LIN {X 0,Y 223.489,Z 613.022,A -85,B 0,C 180,E1 -23403.605,E2 -23403.605} C_VEL
LIN {X 0,Y 223.354,Z 613.371,A -85,B 0,C 180,E1 -23409.051,E2 -23409.051} C_VEL
LIN {X 0,Y 224.233,Z 615.221,A -85,B 0,C 180,E1 -23413.695,E2 -23413.695} C_VEL
LIN {X 0,Y 226.542,Z 620.688,A -85,B 0,C 180,E1 -23419.952,E2 -23419.952} C_VEL
LIN {X 0,Y 227.439,Z 623.666,A -85,B 0,C 180,E1 -23422.032,E2 -23422.032} C_VEL
LIN {X 0,Y 228.456,Z 630.685,A -85,B 0,C 180,E1 -23425.51,E2 -23425.51} C_VEL
LIN {X 0,Y 229.459,Z 640.943,A -85,B 0,C 180,E1 -23429.676,E2 -23429.676} C_VEL
LIN {X 0,Y 229.456,Z 644.838,A -85,B 0,C 180,E1 -23430.955,E2 -23430.955} C_VEL
LIN {X 0,Y 226.429,Z 656.895,A -85,B 0,C 180,E1 -23433.683,E2 -23433.683} C_VEL
LIN {X 0,Y 221.885,Z 669.855,A -85,B 0,C 180,E1 -23436.516,E2 -23436.516} C_VEL
LIN {X 0,Y 214.485,Z 681.955,A -85,B 0,C 180,E1 -23438.563,E2 -23438.563} C_VEL
LIN {X 0,Y 205.907,Z 694.618,A -85,B 0,C 180,E1 -23441.336,E2 -23441.336} C_VEL
LIN {X 0,Y 198.409,Z 704.732,A -85,B 0,C 180,E1 -23444.173,E2 -23444.173} C_VEL
LIN {X 0,Y 190.475,Z 714.65,A -85,B 0,C 180,E1 -23447.682,E2 -23447.682} C_VEL
LIN {X 0,Y 184.311,Z 722.053,A -85,B 0,C 180,E1 -23451.015,E2 -23451.015} C_VEL
LIN {X 0,Y 178.043,Z 729.213,A -85,B 0,C 180,E1 -23455.088,E2 -23455.088} C_VEL
LIN {X 0,Y 172.781,Z 735.226,A -85,B 0,C 180,E1 -23459.443,E2 -23459.443} C_VEL
LIN {X 0,Y 167.694,Z 741.138,A -85,B 0,C 180,E1 -23465.226,E2 -23465.226} C_VEL
LIN {X 0,Y 164.518,Z 745.056,A -85,B 0,C 180,E1 -23470.746,E2 -23470.746} C_VEL
LIN {X 0,Y 163.031,Z 746.186,A -85,B 0,C 180,E1 -23472.711,E2 -23472.711} C_VEL
LIN {X 0,Y 159.183,Z 747.539,A -85,B 0,C 180,E1 -23475.926,E2 -23475.926} C_VEL
LIN {X 0,Y 156.295,Z 748.29,A -85,B 0,C 180,E1 -23478.609,E2 -23478.609} C_VEL
LIN {X 0,Y 155.1,Z 748.716,A -85,B 0,C 180,E1 -23480.741,E2 -23480.741} C_VEL
LIN {X 0,Y 155.005,Z 748.773,A -85,B 0,C 180,E1 -23481.468,E2 -23481.468} C_VEL
LIN {X 0,Y 155.163,Z 749.11,A -85,B 0,C 180,E1 -23485.174,E2 -23485.174} C_VEL
LIN {X 0,Y 155.407,Z 748.7,A -85,B 0,C 180,E1 -23490.003,E2 -23490.003} C_VEL
LIN {X 0,Y 155.267,Z 747.247,A -85,B 0,C 180,E1 -23495.262,E2 -23495.262} C_VEL
LIN {X 0,Y 155.222,Z 744.685,A -85,B 0,C 180,E1 -23500.437,E2 -23500.437} C_VEL
LIN {X 0,Y 156.163,Z 741.06,A -85,B 0,C 180,E1 -23505.668,E2 -23505.668} C_VEL
LIN {X 0,Y 158.061,Z 736.145,A -85,B 0,C 180,E1 -23510.977,E2 -23510.977} C_VEL
LIN {X 0,Y 160.289,Z 731.655,A -85,B 0,C 180,E1 -23514.965,E2 -23514.965} C_VEL
LIN {X 0,Y 165.09,Z 728.65,A -85,B 0,C 180,E1 -23520.723,E2 -23520.723} C_VEL
LIN {X 0,Y 173.61,Z 723.828,A -85,B 0,C 180,E1 -23527.392,E2 -23527.392} C_VEL
LIN {X 0,Y 186.812,Z 716.879,A -85,B 0,C 180,E1 -23534.108,E2 -23534.108} C_VEL
LIN {X 0,Y 199.391,Z 710.477,A -85,B 0,C 180,E1 -23538.657,E2 -23538.657} C_VEL
LIN {X 0,Y 200.155,Z 709.902,A -85,B 0,C 180,E1 -23539.319,E2 -23539.319} C_VEL
LIN {X 0,Y 189.134,Z 711.932,A -85,B 0,C 180,E1 -23543.521,E2 -23543.521} C_VEL
LIN {X 0,Y 178.051,Z 713.204,A -85,B 0,C 180,E1 -23549.128,E2 -23549.128} C_VEL
LIN {X 0,Y 169.257,Z 713.167,A -85,B 0,C 180,E1 -23555.468,E2 -23555.468} C_VEL
LIN {X 0,Y 162.754,Z 711.681,A -85,B 0,C 180,E1 -23562.407,E2 -23562.407} C_VEL
LIN {X 0,Y 159.866,Z 709.778,A -85,B 0,C 180,E1 -23567.303,E2 -23567.303} C_VEL
LIN {X 0,Y 157.754,Z 707.203,A -85,B 0,C 180,E1 -23572.321,E2 -23572.321} C_VEL
LIN {X 0,Y 156.22,Z 701.701,A -85,B 0,C 180,E1 -23580.001,E2 -23580.001} C_VEL
LIN {X 0,Y 156.351,Z 696.898,A -85,B 0,C 180,E1 -23585.159,E2 -23585.159} C_VEL
LIN {X 0,Y 156.849,Z 691.072,A -85,B 0,C 180,E1 -23590.326,E2 -23590.326} C_VEL
LIN {X 0,Y 158.04,Z 684.129,A -85,B 0,C 180,E1 -23595.476,E2 -23595.476} C_VEL
LIN {X 0,Y 160.485,Z 674.694,A -85,B 0,C 180,E1 -23601.18,E2 -23601.18} C_VEL
LIN {X 0,Y 164.064,Z 663.436,A -85,B 0,C 180,E1 -23606.731,E2 -23606.731} C_VEL
LIN {X 0,Y 168.255,Z 651.541,A -85,B 0,C 180,E1 -23611.476,E2 -23611.476} C_VEL
LIN {X 0,Y 173.138,Z 637.728,A -85,B 0,C 180,E1 -23615.982,E2 -23615.982} C_VEL
LIN {X 0,Y 178.436,Z 623.245,A -85,B 0,C 180,E1 -23619.796,E2 -23619.796} C_VEL
LIN {X 0,Y 180.247,Z 618.116,A -85,B 0,C 180,E1 -23620.962,E2 -23620.962} C_VEL
LIN {X 0,Y 180.924,Z 618.131,A -85,B 0,C 180,E1 -23621.329,E2 -23621.329} C_VEL
LIN {X 0,Y 183.088,Z 617.315,A -85,B 0,C 180,E1 -23622.204,E2 -23622.204} C_VEL
LIN {X 0,Y 185.677,Z 615.473,A -85,B 0,C 180,E1 -23622.948,E2 -23622.948} C_VEL
LIN {X 0,Y 189.612,Z 611.812,A -85,B 0,C 180,E1 -23623.859,E2 -23623.859} C_VEL
LIN {X 0,Y 191.1,Z 610.979,A -85,B 0,C 180,E1 -23624.328,E2 -23624.328} C_VEL
LIN {X 0,Y 200.001,Z 609.038,A -85,B 0,C 180,E1 -23627.557,E2 -23627.557} C_VEL
LIN {X 0,Y 202.173,Z 618.005,A -85,B 0,C 180,E1 -23630.328,E2 -23630.328} C_VEL
LIN {X 0,Y 203.073,Z 626.979,A -85,B 0,C 180,E1 -23632.75,E2 -23632.75} C_VEL
LIN {X 0,Y 203.116,Z 633.014,A -85,B 0,C 180,E1 -23634.296,E2 -23634.296} C_VEL
LIN {X 0,Y 197.422,Z 646.866,A -85,B 0,C 180,E1 -23636.508,E2 -23636.508} C_VEL
LIN {X 0,Y 191.451,Z 659.757,A -85,B 0,C 180,E1 -23639.072,E2 -23639.072} C_VEL
LIN {X 0,Y 185.064,Z 672.439,A -85,B 0,C 180,E1 -23642.274,E2 -23642.274} C_VEL
LIN {X 0,Y 179.25,Z 683.136,A -85,B 0,C 180,E1 -23645.687,E2 -23645.687} C_VEL
LIN {X 0,Y 173.819,Z 692.349,A -85,B 0,C 180,E1 -23649.278,E2 -23649.278} C_VEL
LIN {X 0,Y 169.275,Z 700.275,A -85,B 0,C 180,E1 -23653.102,E2 -23653.102} C_VEL
LIN {X 0,Y 164.71,Z 707.873,A -85,B 0,C 180,E1 -23657.679,E2 -23657.679} C_VEL
LIN {X 0,Y 161.077,Z 714.188,A -85,B 0,C 180,E1 -23662.476,E2 -23662.476} C_VEL
LIN {X 0,Y 158.265,Z 719.384,A -85,B 0,C 180,E1 -23667.452,E2 -23667.452} C_VEL
LIN {X 0,Y 156.429,Z 723.388,A -85,B 0,C 180,E1 -23672.572,E2 -23672.572} C_VEL
LIN {X 0,Y 155.289,Z 726.446,A -85,B 0,C 180,E1 -23677.8,E2 -23677.8} C_VEL
LIN {X 0,Y 154.783,Z 728.481,A -85,B 0,C 180,E1 -23683.119,E2 -23683.119} C_VEL
LIN {X 0,Y 154.975,Z 729.558,A -85,B 0,C 180,E1 -23688.505,E2 -23688.505} C_VEL
LIN {X 0,Y 155.836,Z 729.668,A -85,B 0,C 180,E1 -23693.943,E2 -23693.943} C_VEL
LIN {X 0,Y 157.571,Z 728.723,A -85,B 0,C 180,E1 -23699.378,E2 -23699.378} C_VEL
LIN {X 0,Y 160.35,Z 726.79,A -85,B 0,C 180,E1 -23704.731,E2 -23704.731} C_VEL
LIN {X 0,Y 164.191,Z 723.669,A -85,B 0,C 180,E1 -23709.941,E2 -23709.941} C_VEL
LIN {X 0,Y 169.393,Z 719.182,A -85,B 0,C 180,E1 -23715.143,E2 -23715.143} C_VEL
LIN {X 0,Y 175.246,Z 713.903,A -85,B 0,C 180,E1 -23719.633,E2 -23719.633} C_VEL
LIN {X 0,Y 182.399,Z 706.964,A -85,B 0,C 180,E1 -23724.008,E2 -23724.008} C_VEL
LIN {X 0,Y 189.42,Z 699.593,A -85,B 0,C 180,E1 -23727.569,E2 -23727.569} C_VEL
LIN {X 0,Y 197.066,Z 690.909,A -85,B 0,C 180,E1 -23730.892,E2 -23730.892} C_VEL
LIN {X 0,Y 205.336,Z 680.628,A -85,B 0,C 180,E1 -23733.949,E2 -23733.949} C_VEL
LIN {X 0,Y 214.102,Z 668.356,A -85,B 0,C 180,E1 -23736.79,E2 -23736.79} C_VEL
LIN {X 0,Y 221.298,Z 656.932,A -85,B 0,C 180,E1 -23738.883,E2 -23738.883} C_VEL
LIN {X 0,Y 225.042,Z 650.417,A -85,B 0,C 180,E1 -23739.907,E2 -23739.907} C_VEL
LIN {X 0,Y 225.084,Z 646.05,A -85,B 0,C 180,E1 -23741.805,E2 -23741.805} C_VEL
LIN {X 0,Y 224.673,Z 640.373,A -85,B 0,C 180,E1 -23744.579,E2 -23744.579} C_VEL
LIN {X 0,Y 223.711,Z 634.018,A -85,B 0,C 180,E1 -23748.216,E2 -23748.216} C_VEL
LIN {X 0,Y 222.644,Z 628.828,A -85,B 0,C 180,E1 -23751.833,E2 -23751.833} C_VEL
LIN {X 0,Y 221.481,Z 623.917,A -85,B 0,C 180,E1 -23756.361,E2 -23756.361} C_VEL
LIN {X 0,Y 220.778,Z 621.33,A -85,B 0,C 180,E1 -23759.999,E2 -23759.999} C_VEL
LIN {X 0,Y 220.569,Z 619.485,A -85,B 0,C 180,E1 -23763.653,E2 -23763.653} C_VEL
LIN {X 0,Y 220.459,Z 619.877,A -85,B 0,C 180,E1 -23769.171,E2 -23769.171} C_VEL
LIN {X 0,Y 221.087,Z 621.231,A -85,B 0,C 180,E1 -23772.856,E2 -23772.856} C_VEL
LIN {X 0,Y 222.002,Z 624.081,A -85,B 0,C 180,E1 -23776.553,E2 -23776.553} C_VEL
LIN {X 0,Y 223.485,Z 627.57,A -85,B 0,C 180,E1 -23780.237,E2 -23780.237} C_VEL
LIN {X 0,Y 223.819,Z 628.846,A -85,B 0,C 180,E1 -23781.167,E2 -23781.167} C_VEL
LIN {X 0,Y 224.544,Z 635.94,A -85,B 0,C 180,E1 -23784.821,E2 -23784.821} C_VEL
LIN {X 0,Y 225.046,Z 644.518,A -85,B 0,C 180,E1 -23788.484,E2 -23788.484} C_VEL
LIN {X 0,Y 225.04,Z 647.083,A -85,B 0,C 180,E1 -23789.463,E2 -23789.463} C_VEL
LIN {X 0,Y 224.83,Z 648.862,A -85,B 0,C 180,E1 -23790.009,E2 -23790.009} C_VEL
LIN {X 0,Y 221.559,Z 660.162,A -85,B 0,C 180,E1 -23792.632,E2 -23792.632} C_VEL
LIN {X 0,Y 217.114,Z 671.412,A -85,B 0,C 180,E1 -23795.185,E2 -23795.185} C_VEL
LIN {X 0,Y 209.21,Z 683.673,A -85,B 0,C 180,E1 -23797.321,E2 -23797.321} C_VEL
LIN {X 0,Y 201.277,Z 694.886,A -85,B 0,C 180,E1 -23799.814,E2 -23799.814} C_VEL
LIN {X 0,Y 193.488,Z 704.878,A -85,B 0,C 180,E1 -23802.652,E2 -23802.652} C_VEL
LIN {X 0,Y 185.57,Z 714.288,A -85,B 0,C 180,E1 -23806.018,E2 -23806.018} C_VEL
LIN {X 0,Y 178.802,Z 722.034,A -85,B 0,C 180,E1 -23809.572,E2 -23809.572} C_VEL
LIN {X 0,Y 170.689,Z 730.731,A -85,B 0,C 180,E1 -23814.803,E2 -23814.803} C_VEL
LIN {X 0,Y 164.249,Z 737.577,A -85,B 0,C 180,E1 -23820.527,E2 -23820.527} C_VEL
LIN {X 0,Y 159.501,Z 742.743,A -85,B 0,C 180,E1 -23826.64,E2 -23826.64} C_VEL
LIN {X 0,Y 156.926,Z 745.738,A -85,B 0,C 180,E1 -23831.733,E2 -23831.733} C_VEL
LIN {X 0,Y 155.418,Z 747.806,A -85,B 0,C 180,E1 -23836.935,E2 -23836.935} C_VEL
LIN {X 0,Y 155.005,Z 748.773,A -85,B 0,C 180,E1 -23841.468,E2 -23841.468} C_VEL
LIN {X 0,Y 154.379,Z 749.017,A -85,B 0,C 180,E1 -23843.64,E2 -23843.64} C_VEL
LIN {X 0,Y 152.898,Z 748.974,A -85,B 0,C 180,E1 -23845.787,E2 -23845.787} C_VEL
LIN {X 0,Y 148.562,Z 747.904,A -85,B 0,C 180,E1 -23851.659,E2 -23851.659} C_VEL
LIN {X 0,Y 148.205,Z 747.43,A -85,B 0,C 180,E1 -23853.196,E2 -23853.196} C_VEL
LIN {X 0,Y 148.17,Z 746.707,A -85,B 0,C 180,E1 -23855.446,E2 -23855.446} C_VEL
LIN {X 0,Y 148.186,Z 744.082,A -85,B 0,C 180,E1 -23860.938,E2 -23860.938} C_VEL
LIN {X 0,Y 149.659,Z 739.281,A -85,B 0,C 180,E1 -23867.775,E2 -23867.775} C_VEL
LIN {X 0,Y 151.942,Z 734.123,A -85,B 0,C 180,E1 -23873.154,E2 -23873.154} C_VEL
LIN {X 0,Y 153.762,Z 730.941,A -85,B 0,C 180,E1 -23876.102,E2 -23876.102} C_VEL
LIN {X 0,Y 161.607,Z 726.826,A -85,B 0,C 180,E1 -23884.429,E2 -23884.429} C_VEL
LIN {X 0,Y 171.546,Z 722.041,A -85,B 0,C 180,E1 -23890.96,E2 -23890.96} C_VEL
LIN {X 0,Y 184.2,Z 716.172,A -85,B 0,C 180,E1 -23896.626,E2 -23896.626} C_VEL
LIN {X 0,Y 190.089,Z 713.503,A -85,B 0,C 180,E1 -23898.714,E2 -23898.714} C_VEL
LIN {X 0,Y 190.869,Z 712.92,A -85,B 0,C 180,E1 -23899.48,E2 -23899.48} C_VEL
LIN {X 0,Y 179.634,Z 714.285,A -85,B 0,C 180,E1 -23904.067,E2 -23904.067} C_VEL
LIN {X 0,Y 168.819,Z 714.719,A -85,B 0,C 180,E1 -23910.03,E2 -23910.03} C_VEL
LIN {X 0,Y 160.341,Z 713.845,A -85,B 0,C 180,E1 -23916.767,E2 -23916.767} C_VEL
LIN {X 0,Y 154.361,Z 711.482,A -85,B 0,C 180,E1 -23924.148,E2 -23924.148} C_VEL
LIN {X 0,Y 151.752,Z 709.006,A -85,B 0,C 180,E1 -23929.326,E2 -23929.326} C_VEL
LIN {X 0,Y 149.904,Z 705.812,A -85,B 0,C 180,E1 -23934.621,E2 -23934.621} C_VEL
LIN {X 0,Y 149.08,Z 700.566,A -85,B 0,C 180,E1 -23941.352,E2 -23941.352} C_VEL
LIN {X 0,Y 149.332,Z 695.303,A -85,B 0,C 180,E1 -23946.758,E2 -23946.758} C_VEL
LIN {X 0,Y 150.076,Z 689,A -85,B 0,C 180,E1 -23952.167,E2 -23952.167} C_VEL
LIN {X 0,Y 151.833,Z 680.442,A -85,B 0,C 180,E1 -23958.208,E2 -23958.208} C_VEL
LIN {X 0,Y 154.571,Z 671.347,A -85,B 0,C 180,E1 -23963.445,E2 -23963.445} C_VEL
LIN {X 0,Y 158.134,Z 660.693,A -85,B 0,C 180,E1 -23968.541,E2 -23968.541} C_VEL
LIN {X 0,Y 162.689,Z 648.26,A -85,B 0,C 180,E1 -23973.422,E2 -23973.422} C_VEL
LIN {X 0,Y 167.242,Z 635.959,A -85,B 0,C 180,E1 -23977.391,E2 -23977.391} C_VEL
LIN {X 0,Y 169.446,Z 630.318,A -85,B 0,C 180,E1 -23979.046,E2 -23979.046} C_VEL
LIN {X 0,Y 170.577,Z 630.187,A -85,B 0,C 180,E1 -23979.69,E2 -23979.69} C_VEL
LIN {X 0,Y 172.808,Z 629.111,A -85,B 0,C 180,E1 -23980.597,E2 -23980.597} C_VEL
LIN {X 0,Y 176.713,Z 626.375,A -85,B 0,C 180,E1 -23981.773,E2 -23981.773} C_VEL
LIN {X 0,Y 178.152,Z 625.177,A -85,B 0,C 180,E1 -23982.118,E2 -23982.118} C_VEL
LIN {X 0,Y 183.046,Z 622.498,A -85,B 0,C 180,E1 -23983.719,E2 -23983.719} C_VEL
LIN {X 0,Y 187.136,Z 619.45,A -85,B 0,C 180,E1 -23984.764,E2 -23984.764} C_VEL
LIN {X 0,Y 188.591,Z 618.221,A -85,B 0,C 180,E1 -23985.078,E2 -23985.078} C_VEL
LIN {X 0,Y 193.37,Z 616.385,A -85,B 0,C 180,E1 -23986.628,E2 -23986.628} C_VEL
LIN {X 0,Y 195.642,Z 615.928,A -85,B 0,C 180,E1 -23987.428,E2 -23987.428} C_VEL
LIN {X 0,Y 196.622,Z 619.354,A -85,B 0,C 180,E1 -23988.645,E2 -23988.645} C_VEL
LIN {X 0,Y 197.469,Z 625.794,A -85,B 0,C 180,E1 -23990.579,E2 -23990.579} C_VEL
LIN {X 0,Y 197.745,Z 633.888,A -85,B 0,C 180,E1 -23992.827,E2 -23992.827} C_VEL
LIN {X 0,Y 196.896,Z 636.565,A -85,B 0,C 180,E1 -23993.28,E2 -23993.28} C_VEL
LIN {X 0,Y 190.573,Z 651.082,A -85,B 0,C 180,E1 -23995.776,E2 -23995.776} C_VEL
LIN {X 0,Y 184.485,Z 663.343,A -85,B 0,C 180,E1 -23998.41,E2 -23998.41} C_VEL
LIN {X 0,Y 177.966,Z 675.514,A -85,B 0,C 180,E1 -24001.711,E2 -24001.711} C_VEL
LIN {X 0,Y 172.001,Z 685.898,A -85,B 0,C 180,E1 -24005.238,E2 -24005.238} C_VEL
LIN {X 0,Y 165.764,Z 695.986,A -85,B 0,C 180,E1 -24009.524,E2 -24009.524} C_VEL
LIN {X 0,Y 161.111,Z 703.593,A -85,B 0,C 180,E1 -24013.68,E2 -24013.68} C_VEL
LIN {X 0,Y 156.765,Z 710.557,A -85,B 0,C 180,E1 -24018.359,E2 -24018.359} C_VEL
LIN {X 0,Y 153.221,Z 716.506,A -85,B 0,C 180,E1 -24023.413,E2 -24023.413} C_VEL
LIN {X 0,Y 150.114,Z 722.307,A -85,B 0,C 180,E1 -24029.997,E2 -24029.997} C_VEL
LIN {X 0,Y 148.488,Z 726.191,A -85,B 0,C 180,E1 -24036.3,E2 -24036.3} C_VEL
LIN {X 0,Y 147.829,Z 728.225,A -85,B 0,C 180,E1 -24040.959,E2 -24040.959} C_VEL
LIN {X 0,Y 147.753,Z 729.674,A -85,B 0,C 180,E1 -24046.579,E2 -24046.579} C_VEL
LIN {X 0,Y 148.348,Z 730.206,A -85,B 0,C 180,E1 -24052.268,E2 -24052.268} C_VEL
LIN {X 0,Y 149.877,Z 729.71,A -85,B 0,C 180,E1 -24057.961,E2 -24057.961} C_VEL
LIN {X 0,Y 152.731,Z 727.977,A -85,B 0,C 180,E1 -24064.076,E2 -24064.076} C_VEL
LIN {X 0,Y 156.109,Z 725.6,A -85,B 0,C 180,E1 -24069.066,E2 -24069.066} C_VEL
LIN {X 0,Y 162.176,Z 720.844,A -85,B 0,C 180,E1 -24075.44,E2 -24075.44} C_VEL
LIN {X 0,Y 168.647,Z 715.369,A -85,B 0,C 180,E1 -24080.434,E2 -24080.434} C_VEL
LIN {X 0,Y 176.015,Z 708.671,A -85,B 0,C 180,E1 -24084.933,E2 -24084.933} C_VEL
LIN {X 0,Y 184.328,Z 700.456,A -85,B 0,C 180,E1 -24089.073,E2 -24089.073} C_VEL
LIN {X 0,Y 192.282,Z 691.867,A -85,B 0,C 180,E1 -24092.412,E2 -24092.412} C_VEL
LIN {X 0,Y 200.84,Z 681.65,A -85,B 0,C 180,E1 -24095.474,E2 -24095.474} C_VEL
LIN {X 0,Y 208.184,Z 671.874,A -85,B 0,C 180,E1 -24097.794,E2 -24097.794} C_VEL
LIN {X 0,Y 215.952,Z 660.423,A -85,B 0,C 180,E1 -24099.996,E2 -24099.996} C_VEL
LIN {X 0,Y 219.532,Z 654.659,A -85,B 0,C 180,E1 -24100.938,E2 -24100.938} C_VEL
LIN {X 0,Y 220.2,Z 652.915,A -85,B 0,C 180,E1 -24101.387,E2 -24101.387} C_VEL
LIN {X 0,Y 220.25,Z 647.016,A -85,B 0,C 180,E1 -24104.262,E2 -24104.262} C_VEL
LIN {X 0,Y 219.848,Z 642.047,A -85,B 0,C 180,E1 -24107.068,E2 -24107.068} C_VEL
LIN {X 0,Y 219.123,Z 636.488,A -85,B 0,C 180,E1 -24110.771,E2 -24110.771} C_VEL
LIN {X 0,Y 218.552,Z 633.135,A -85,B 0,C 180,E1 -24113.537,E2 -24113.537} C_VEL
LIN {X 0,Y 218.036,Z 630.331,A -85,B 0,C 180,E1 -24116.303,E2 -24116.303} C_VEL
LIN {X 0,Y 217.543,Z 627.695,A -85,B 0,C 180,E1 -24119.999,E2 -24119.999} C_VEL
LIN {X 0,Y 217.4,Z 625.859,A -85,B 0,C 180,E1 -24123.706,E2 -24123.706} C_VEL
LIN {X 0,Y 217.358,Z 626.302,A -85,B 0,C 180,E1 -24129.303,E2 -24129.303} C_VEL
LIN {X 0,Y 217.941,Z 627.789,A -85,B 0,C 180,E1 -24133.045,E2 -24133.045} C_VEL
LIN {X 0,Y 218.808,Z 630.672,A -85,B 0,C 180,E1 -24136.802,E2 -24136.802} C_VEL
LIN {X 0,Y 219.727,Z 632.927,A -85,B 0,C 180,E1 -24139.256,E2 -24139.256} C_VEL
LIN {X 0,Y 220.142,Z 634.473,A -85,B 0,C 180,E1 -24140.558,E2 -24140.558} C_VEL
LIN {X 0,Y 220.49,Z 640.824,A -85,B 0,C 180,E1 -24143.978,E2 -24143.978} C_VEL
LIN {X 0,Y 220.592,Z 649.938,A -85,B 0,C 180,E1 -24148.028,E2 -24148.028} C_VEL
LIN {X 0,Y 220.209,Z 652.857,A -85,B 0,C 180,E1 -24149.028,E2 -24149.028} C_VEL
LIN {X 0,Y 216.478,Z 663.697,A -85,B 0,C 180,E1 -24151.632,E2 -24151.632} C_VEL
LIN {X 0,Y 212.462,Z 672.993,A -85,B 0,C 180,E1 -24153.792,E2 -24153.792} C_VEL
LIN {X 0,Y 204.686,Z 684.456,A -85,B 0,C 180,E1 -24155.827,E2 -24155.827} C_VEL
LIN {X 0,Y 196.796,Z 695.125,A -85,B 0,C 180,E1 -24158.222,E2 -24158.222} C_VEL
LIN {X 0,Y 187.623,Z 706.369,A -85,B 0,C 180,E1 -24161.486,E2 -24161.486} C_VEL
LIN {X 0,Y 179.119,Z 715.833,A -85,B 0,C 180,E1 -24165.073,E2 -24165.073} C_VEL
LIN {X 0,Y 171.525,Z 723.841,A -85,B 0,C 180,E1 -24169.04,E2 -24169.04} C_VEL
LIN {X 0,Y 164.864,Z 730.604,A -85,B 0,C 180,E1 -24173.362,E2 -24173.362} C_VEL
LIN {X 0,Y 157.986,Z 737.372,A -85,B 0,C 180,E1 -24179.235,E2 -24179.235} C_VEL
LIN {X 0,Y 152.895,Z 742.475,A -85,B 0,C 180,E1 -24185.566,E2 -24185.566} C_VEL
LIN {X 0,Y 150.109,Z 745.398,A -85,B 0,C 180,E1 -24190.872,E2 -24190.872} C_VEL
LIN {X 0,Y 148.425,Z 747.432,A -85,B 0,C 180,E1 -24196.308,E2 -24196.308} C_VEL
LIN {X 0,Y 147.935,Z 748.453,A -85,B 0,C 180,E1 -24201.809,E2 -24201.809} C_VEL
LIN {X 0,Y 148.08,Z 748.629,A -85,B 0,C 180,E1 -24205.315,E2 -24205.315} C_VEL
LIN {X 0,Y 148.34,Z 748.202,A -85,B 0,C 180,E1 -24210.003,E2 -24210.003} C_VEL
LIN {X 0,Y 148.205,Z 747.43,A -85,B 0,C 180,E1 -24213.196,E2 -24213.196} C_VEL
LIN {X 0,Y 147.436,Z 746.663,A -85,B 0,C 180,E1 -24215.438,E2 -24215.438} C_VEL
LIN {X 0,Y 144.551,Z 744.902,A -85,B 0,C 180,E1 -24219.095,E2 -24219.095} C_VEL
LIN {X 0,Y 142.342,Z 743.201,A -85,B 0,C 180,E1 -24222.094,E2 -24222.094} C_VEL
LIN {X 0,Y 141.682,Z 741.692,A -85,B 0,C 180,E1 -24224.414,E2 -24224.414} C_VEL
LIN {X 0,Y 141.778,Z 741.182,A -85,B 0,C 180,E1 -24225.192,E2 -24225.192} C_VEL
LIN {X 0,Y 143.322,Z 737.404,A -85,B 0,C 180,E1 -24230.078,E2 -24230.078} C_VEL
LIN {X 0,Y 146.163,Z 731.888,A -85,B 0,C 180,E1 -24235.645,E2 -24235.645} C_VEL
LIN {X 0,Y 147.333,Z 730.153,A -85,B 0,C 180,E1 -24237.334,E2 -24237.334} C_VEL
LIN {X 0,Y 154.789,Z 726.854,A -85,B 0,C 180,E1 -24245.19,E2 -24245.19} C_VEL
LIN {X 0,Y 166.205,Z 721.991,A -85,B 0,C 180,E1 -24252.578,E2 -24252.578} C_VEL
LIN {X 0,Y 180.789,Z 716.05,A -85,B 0,C 180,E1 -24258.769,E2 -24258.769} C_VEL
LIN {X 0,Y 181.54,Z 715.474,A -85,B 0,C 180,E1 -24259.647,E2 -24259.647} C_VEL
LIN {X 0,Y 170.099,Z 716.149,A -85,B 0,C 180,E1 -24264.66,E2 -24264.66} C_VEL
LIN {X 0,Y 162.82,Z 716.042,A -85,B 0,C 180,E1 -24268.805,E2 -24268.805} C_VEL
LIN {X 0,Y 153.899,Z 714.772,A -85,B 0,C 180,E1 -24275.734,E2 -24275.734} C_VEL
LIN {X 0,Y 149.359,Z 713.166,A -85,B 0,C 180,E1 -24280.77,E2 -24280.77} C_VEL
LIN {X 0,Y 144.787,Z 709.4,A -85,B 0,C 180,E1 -24288.806,E2 -24288.806} C_VEL
LIN {X 0,Y 142.299,Z 703.903,A -85,B 0,C 180,E1 -24297.17,E2 -24297.17} C_VEL
LIN {X 0,Y 142.115,Z 697.855,A -85,B 0,C 180,E1 -24304.255,E2 -24304.255} C_VEL
LIN {X 0,Y 142.819,Z 690.204,A -85,B 0,C 180,E1 -24311.353,E2 -24311.353} C_VEL
LIN {X 0,Y 144.486,Z 681.679,A -85,B 0,C 180,E1 -24317.7,E2 -24317.7} C_VEL
LIN {X 0,Y 147.108,Z 672.694,A -85,B 0,C 180,E1 -24323.214,E2 -24323.214} C_VEL
LIN {X 0,Y 150.757,Z 662.199,A -85,B 0,C 180,E1 -24328.546,E2 -24328.546} C_VEL
LIN {X 0,Y 155.392,Z 649.876,A -85,B 0,C 180,E1 -24333.646,E2 -24333.646} C_VEL
LIN {X 0,Y 158.706,Z 641.127,A -85,B 0,C 180,E1 -24336.789,E2 -24336.789} C_VEL
LIN {X 0,Y 160.394,Z 640.817,A -85,B 0,C 180,E1 -24337.84,E2 -24337.84} C_VEL
LIN {X 0,Y 162.587,Z 639.739,A -85,B 0,C 180,E1 -24338.814,E2 -24338.814} C_VEL
LIN {X 0,Y 167.748,Z 636.226,A -85,B 0,C 180,E1 -24340.497,E2 -24340.497} C_VEL
LIN {X 0,Y 169.961,Z 635.352,A -85,B 0,C 180,E1 -24341.424,E2 -24341.424} C_VEL
LIN {X 0,Y 172.386,Z 634.118,A -85,B 0,C 180,E1 -24342.276,E2 -24342.276} C_VEL
LIN {X 0,Y 176.477,Z 631.399,A -85,B 0,C 180,E1 -24343.392,E2 -24343.392} C_VEL
LIN {X 0,Y 177.913,Z 630.272,A -85,B 0,C 180,E1 -24343.734,E2 -24343.734} C_VEL
LIN {X 0,Y 182.982,Z 627.571,A -85,B 0,C 180,E1 -24345.281,E2 -24345.281} C_VEL
LIN {X 0,Y 188.642,Z 623.693,A -85,B 0,C 180,E1 -24346.594,E2 -24346.594} C_VEL
LIN {X 0,Y 191.092,Z 622.815,A -85,B 0,C 180,E1 -24347.356,E2 -24347.356} C_VEL
LIN {X 0,Y 191.778,Z 624.167,A -85,B 0,C 180,E1 -24348.016,E2 -24348.016} C_VEL
LIN {X 0,Y 192.285,Z 631.101,A -85,B 0,C 180,E1 -24350.136,E2 -24350.136} C_VEL
LIN {X 0,Y 192.307,Z 636.049,A -85,B 0,C 180,E1 -24351.588,E2 -24351.588} C_VEL
LIN {X 0,Y 186.942,Z 648.413,A -85,B 0,C 180,E1 -24353.691,E2 -24353.691} C_VEL
LIN {X 0,Y 180.544,Z 661.203,A -85,B 0,C 180,E1 -24356.307,E2 -24356.307} C_VEL
LIN {X 0,Y 174.638,Z 672.113,A -85,B 0,C 180,E1 -24359.127,E2 -24359.127} C_VEL
LIN {X 0,Y 168.256,Z 683.004,A -85,B 0,C 180,E1 -24362.645,E2 -24362.645} C_VEL
LIN {X 0,Y 162.281,Z 692.393,A -85,B 0,C 180,E1 -24366.382,E2 -24366.382} C_VEL
LIN {X 0,Y 157.102,Z 700.423,A -85,B 0,C 180,E1 -24370.394,E2 -24370.394} C_VEL
LIN {X 0,Y 152.019,Z 708.15,A -85,B 0,C 180,E1 -24375.267,E2 -24375.267} C_VEL
LIN {X 0,Y 147.88,Z 714.597,A -85,B 0,C 180,E1 -24380.422,E2 -24380.422} C_VEL
LIN {X 0,Y 144.692,Z 719.857,A -85,B 0,C 180,E1 -24385.819,E2 -24385.819} C_VEL
LIN {X 0,Y 142.987,Z 723.08,A -85,B 0,C 180,E1 -24389.997,E2 -24389.997} C_VEL
LIN {X 0,Y 141.399,Z 726.686,A -85,B 0,C 180,E1 -24396.233,E2 -24396.233} C_VEL
LIN {X 0,Y 140.676,Z 728.817,A -85,B 0,C 180,E1 -24401.524,E2 -24401.524} C_VEL
LIN {X 0,Y 140.729,Z 730.218,A -85,B 0,C 180,E1 -24407.432,E2 -24407.432} C_VEL
LIN {X 0,Y 141.465,Z 730.65,A -85,B 0,C 180,E1 -24413.415,E2 -24413.415} C_VEL
LIN {X 0,Y 143.27,Z 730.105,A -85,B 0,C 180,E1 -24419.372,E2 -24419.372} C_VEL
LIN {X 0,Y 146.163,Z 728.457,A -85,B 0,C 180,E1 -24425.236,E2 -24425.236} C_VEL
LIN {X 0,Y 151.138,Z 725.132,A -85,B 0,C 180,E1 -24431.924,E2 -24431.924} C_VEL
LIN {X 0,Y 157.638,Z 720.32,A -85,B 0,C 180,E1 -24438.028,E2 -24438.028} C_VEL
LIN {X 0,Y 163.773,Z 715.452,A -85,B 0,C 180,E1 -24442.424,E2 -24442.424} C_VEL
LIN {X 0,Y 171.721,Z 708.54,A -85,B 0,C 180,E1 -24447.029,E2 -24447.029} C_VEL
LIN {X 0,Y 180.526,Z 700.19,A -85,B 0,C 180,E1 -24451.15,E2 -24451.15} C_VEL
LIN {X 0,Y 188.864,Z 691.443,A -85,B 0,C 180,E1 -24454.468,E2 -24454.468} C_VEL
LIN {X 0,Y 197.811,Z 681.113,A -85,B 0,C 180,E1 -24457.473,E2 -24457.473} C_VEL
LIN {X 0,Y 206.719,Z 669.422,A -85,B 0,C 180,E1 -24460.124,E2 -24460.124} C_VEL
LIN {X 0,Y 214.168,Z 658.376,A -85,B 0,C 180,E1 -24462.101,E2 -24462.101} C_VEL
LIN {X 0,Y 215.3,Z 656.539,A -85,B 0,C 180,E1 -24462.425,E2 -24462.425} C_VEL
LIN {X 0,Y 215.53,Z 651.771,A -85,B 0,C 180,E1 -24464.878,E2 -24464.878} C_VEL
LIN {X 0,Y 215.355,Z 646.218,A -85,B 0,C 180,E1 -24468.234,E2 -24468.234} C_VEL
LIN {X 0,Y 215.014,Z 641.631,A -85,B 0,C 180,E1 -24471.541,E2 -24471.541} C_VEL
LIN {X 0,Y 214.583,Z 638.444,A -85,B 0,C 180,E1 -24474.36,E2 -24474.36} C_VEL
LIN {X 0,Y 214.215,Z 635.145,A -85,B 0,C 180,E1 -24478.119,E2 -24478.119} C_VEL
LIN {X 0,Y 213.967,Z 632.931,A -85,B 0,C 180,E1 -24481.881,E2 -24481.881} C_VEL
LIN {X 0,Y 214.049,Z 632.115,A -85,B 0,C 180,E1 -24483.764,E2 -24483.764} C_VEL
LIN {X 0,Y 213.916,Z 632.273,A -85,B 0,C 180,E1 -24487.551,E2 -24487.551} C_VEL
LIN {X 0,Y 214.272,Z 633.3,A -85,B 0,C 180,E1 -24491.349,E2 -24491.349} C_VEL
LIN {X 0,Y 214.593,Z 634.241,A -85,B 0,C 180,E1 -24493.252,E2 -24493.252} C_VEL
LIN {X 0,Y 216.025,Z 638.9,A -85,B 0,C 180,E1 -24498.985,E2 -24498.985} C_VEL
LIN {X 0,Y 216.257,Z 639.924,A -85,B 0,C 180,E1 -24499.852,E2 -24499.852} C_VEL
LIN {X 0,Y 216.338,Z 645.255,A -85,B 0,C 180,E1 -24502.943,E2 -24502.943} C_VEL
LIN {X 0,Y 216.035,Z 654.103,A -85,B 0,C 180,E1 -24507.093,E2 -24507.093} C_VEL
LIN {X 0,Y 215.908,Z 655.441,A -85,B 0,C 180,E1 -24507.635,E2 -24507.635} C_VEL
LIN {X 0,Y 213.654,Z 661.821,A -85,B 0,C 180,E1 -24509.277,E2 -24509.277} C_VEL
LIN {X 0,Y 210.36,Z 669.463,A -85,B 0,C 180,E1 -24511.122,E2 -24511.122} C_VEL
LIN {X 0,Y 207.924,Z 674.527,A -85,B 0,C 180,E1 -24512.331,E2 -24512.331} C_VEL
LIN {X 0,Y 199.074,Z 686.98,A -85,B 0,C 180,E1 -24514.635,E2 -24514.635} C_VEL
LIN {X 0,Y 190.019,Z 698.298,A -85,B 0,C 180,E1 -24517.331,E2 -24517.331} C_VEL
LIN {X 0,Y 180.684,Z 708.952,A -85,B 0,C 180,E1 -24520.674,E2 -24520.674} C_VEL
LIN {X 0,Y 172.082,Z 717.977,A -85,B 0,C 180,E1 -24524.384,E2 -24524.384} C_VEL
LIN {X 0,Y 164.305,Z 725.607,A -85,B 0,C 180,E1 -24528.475,E2 -24528.475} C_VEL
LIN {X 0,Y 155.929,Z 733.435,A -85,B 0,C 180,E1 -24534.221,E2 -24534.221} C_VEL
LIN {X 0,Y 149.395,Z 739.354,A -85,B 0,C 180,E1 -24540.403,E2 -24540.403} C_VEL
LIN {X 0,Y 146.351,Z 742.199,A -85,B 0,C 180,E1 -24544.397,E2 -24544.397} C_VEL
LIN {X 0,Y 143.329,Z 745.059,A -85,B 0,C 180,E1 -24549.929,E2 -24549.929} C_VEL
LIN {X 0,Y 141.45,Z 747.052,A -85,B 0,C 180,E1 -24555.619,E2 -24555.619} C_VEL
LIN {X 0,Y 140.856,Z 748.013,A -85,B 0,C 180,E1 -24561.395,E2 -24561.395} C_VEL
LIN {X 0,Y 141.081,Z 748.099,A -85,B 0,C 180,E1 -24567.148,E2 -24567.148} C_VEL
LIN {X 0,Y 141.274,Z 747.702,A -85,B 0,C 180,E1 -24570.003,E2 -24570.003} C_VEL
LIN {X 0,Y 141.1,Z 746.41,A -85,B 0,C 180,E1 -24575.029,E2 -24575.029} C_VEL
LIN {X 0,Y 141.142,Z 743.47,A -85,B 0,C 180,E1 -24581.492,E2 -24581.492} C_VEL
LIN {X 0,Y 141.778,Z 741.182,A -85,B 0,C 180,E1 -24585.192,E2 -24585.192} C_VEL
LIN {X 0,Y 141.734,Z 739.589,A -85,B 0,C 180,E1 -24587.492,E2 -24587.492} C_VEL
LIN {X 0,Y 140.196,Z 736.568,A -85,B 0,C 180,E1 -24591.287,E2 -24591.287} C_VEL
LIN {X 0,Y 139.209,Z 733.803,A -85,B 0,C 180,E1 -24594.331,E2 -24594.331} C_VEL
LIN {X 0,Y 139.52,Z 731.506,A -85,B 0,C 180,E1 -24596.577,E2 -24596.577} C_VEL
LIN {X 0,Y 139.939,Z 730.702,A -85,B 0,C 180,E1 -24597.298,E2 -24597.298} C_VEL
LIN {X 0,Y 140.993,Z 729.321,A -85,B 0,C 180,E1 -24598.674,E2 -24598.674} C_VEL
LIN {X 0,Y 149.952,Z 725.938,A -85,B 0,C 180,E1 -24607.541,E2 -24607.541} C_VEL
LIN {X 0,Y 161.014,Z 721.927,A -85,B 0,C 180,E1 -24614.3,E2 -24614.3} C_VEL
LIN {X 0,Y 173.065,Z 717.502,A -85,B 0,C 180,E1 -24619.479,E2 -24619.479} C_VEL
LIN {X 0,Y 160.505,Z 717.528,A -85,B 0,C 180,E1 -24625.305,E2 -24625.305} C_VEL
LIN {X 0,Y 150.347,Z 716.303,A -85,B 0,C 180,E1 -24632.132,E2 -24632.132} C_VEL
LIN {X 0,Y 142.694,Z 713.729,A -85,B 0,C 180,E1 -24639.834,E2 -24639.834} C_VEL
LIN {X 0,Y 139.199,Z 711.181,A -85,B 0,C 180,E1 -24645.379,E2 -24645.379} C_VEL
LIN {X 0,Y 136.692,Z 707.926,A -85,B 0,C 180,E1 -24651.128,E2 -24651.128} C_VEL
LIN {X 0,Y 135.035,Z 702.698,A -85,B 0,C 180,E1 -24658.51,E2 -24658.51} C_VEL
LIN {X 0,Y 135.046,Z 697.503,A -85,B 0,C 180,E1 -24664.479,E2 -24664.479} C_VEL
LIN {X 0,Y 135.557,Z 691.303,A -85,B 0,C 180,E1 -24670.455,E2 -24670.455} C_VEL
LIN {X 0,Y 136.893,Z 683.881,A -85,B 0,C 180,E1 -24676.403,E2 -24676.403} C_VEL
LIN {X 0,Y 139.717,Z 673.974,A -85,B 0,C 180,E1 -24682.946,E2 -24682.946} C_VEL
LIN {X 0,Y 143.389,Z 663.468,A -85,B 0,C 180,E1 -24688.606,E2 -24688.606} C_VEL
LIN {X 0,Y 148.566,Z 650.516,A -85,B 0,C 180,E1 -24694.384,E2 -24694.384} C_VEL
LIN {X 0,Y 152.539,Z 649.199,A -85,B 0,C 180,E1 -24696.797,E2 -24696.797} C_VEL
LIN {X 0,Y 157.209,Z 646.63,A -85,B 0,C 180,E1 -24698.747,E2 -24698.747} C_VEL
LIN {X 0,Y 160.426,Z 645.272,A -85,B 0,C 180,E1 -24700.188,E2 -24700.188} C_VEL
LIN {X 0,Y 167.036,Z 641.397,A -85,B 0,C 180,E1 -24702.316,E2 -24702.316} C_VEL
LIN {X 0,Y 172.018,Z 639.03,A -85,B 0,C 180,E1 -24703.993,E2 -24703.993} C_VEL
LIN {X 0,Y 177.662,Z 635.31,A -85,B 0,C 180,E1 -24705.403,E2 -24705.403} C_VEL
LIN {X 0,Y 182.991,Z 632.549,A -85,B 0,C 180,E1 -24706.864,E2 -24706.864} C_VEL
LIN {X 0,Y 185.877,Z 630.745,A -85,B 0,C 180,E1 -24707.503,E2 -24707.503} C_VEL
LIN {X 0,Y 186.997,Z 630.624,A -85,B 0,C 180,E1 -24707.927,E2 -24707.927} C_VEL
LIN {X 0,Y 186.961,Z 638.195,A -85,B 0,C 180,E1 -24710.277,E2 -24710.277} C_VEL
LIN {X 0,Y 180.232,Z 652.596,A -85,B 0,C 180,E1 -24712.811,E2 -24712.811} C_VEL
LIN {X 0,Y 173.692,Z 664.763,A -85,B 0,C 180,E1 -24715.493,E2 -24715.493} C_VEL
LIN {X 0,Y 166.652,Z 676.854,A -85,B 0,C 180,E1 -24718.893,E2 -24718.893} C_VEL
LIN {X 0,Y 160.196,Z 687.165,A -85,B 0,C 180,E1 -24722.568,E2 -24722.568} C_VEL
LIN {X 0,Y 154.157,Z 696.04,A -85,B 0,C 180,E1 -24726.487,E2 -24726.487} C_VEL
LIN {X 0,Y 149.112,Z 703.548,A -85,B 0,C 180,E1 -24730.733,E2 -24730.733} C_VEL
LIN {X 0,Y 144.015,Z 710.892,A -85,B 0,C 180,E1 -24735.874,E2 -24735.874} C_VEL
LIN {X 0,Y 139.97,Z 716.907,A -85,B 0,C 180,E1 -24741.333,E2 -24741.333} C_VEL
LIN {X 0,Y 136.902,Z 721.774,A -85,B 0,C 180,E1 -24747.054,E2 -24747.054} C_VEL
LIN {X 0,Y 134.945,Z 725.619,A -85,B 0,C 180,E1 -24752.982,E2 -24752.982} C_VEL
LIN {X 0,Y 133.821,Z 728.369,A -85,B 0,C 180,E1 -24759.062,E2 -24759.062} C_VEL
LIN {X 0,Y 133.504,Z 730.224,A -85,B 0,C 180,E1 -24765.257,E2 -24765.257} C_VEL
LIN {X 0,Y 133.752,Z 730.852,A -85,B 0,C 180,E1 -24768.945,E2 -24768.945} C_VEL
LIN {X 0,Y 134.634,Z 731.096,A -85,B 0,C 180,E1 -24774.68,E2 -24774.68} C_VEL
LIN {X 0,Y 136.717,Z 730.486,A -85,B 0,C 180,E1 -24780.93,E2 -24780.93} C_VEL
LIN {X 0,Y 140.014,Z 728.747,A -85,B 0,C 180,E1 -24787.033,E2 -24787.033} C_VEL
LIN {X 0,Y 144.99,Z 725.672,A -85,B 0,C 180,E1 -24793.356,E2 -24793.356} C_VEL
LIN {X 0,Y 150.362,Z 722.039,A -85,B 0,C 180,E1 -24798.399,E2 -24798.399} C_VEL
LIN {X 0,Y 158.819,Z 715.755,A -85,B 0,C 180,E1 -24804.361,E2 -24804.361} C_VEL
LIN {X 0,Y 167.618,Z 708.484,A -85,B 0,C 180,E1 -24809.176,E2 -24809.176} C_VEL
LIN {X 0,Y 175.758,Z 701.07,A -85,B 0,C 180,E1 -24812.83,E2 -24812.83} C_VEL
LIN {X 0,Y 184.419,Z 692.412,A -85,B 0,C 180,E1 -24816.144,E2 -24816.144} C_VEL
LIN {X 0,Y 193.835,Z 681.976,A -85,B 0,C 180,E1 -24819.182,E2 -24819.182} C_VEL
LIN {X 0,Y 203.294,Z 670,A -85,B 0,C 180,E1 -24821.871,E2 -24821.871} C_VEL
LIN {X 0,Y 210.461,Z 659.676,A -85,B 0,C 180,E1 -24823.73,E2 -24823.73} C_VEL
LIN {X 0,Y 210.843,Z 654.811,A -85,B 0,C 180,E1 -24826.506,E2 -24826.506} C_VEL
LIN {X 0,Y 210.88,Z 650.396,A -85,B 0,C 180,E1 -24829.437,E2 -24829.437} C_VEL
LIN {X 0,Y 210.7,Z 645.566,A -85,B 0,C 180,E1 -24833.295,E2 -24833.295} C_VEL
LIN {X 0,Y 210.527,Z 642.816,A -85,B 0,C 180,E1 -24836.171,E2 -24836.171} C_VEL
LIN {X 0,Y 210.336,Z 640.055,A -85,B 0,C 180,E1 -24839.999,E2 -24839.999} C_VEL
LIN {X 0,Y 210.5,Z 638.283,A -85,B 0,C 180,E1 -24843.828,E2 -24843.828} C_VEL
LIN {X 0,Y 210.42,Z 638.473,A -85,B 0,C 180,E1 -24847.677,E2 -24847.677} C_VEL
LIN {X 0,Y 210.772,Z 639.568,A -85,B 0,C 180,E1 -24851.54,E2 -24851.54} C_VEL
LIN {X 0,Y 211.299,Z 641.908,A -85,B 0,C 180,E1 -24855.308,E2 -24855.308} C_VEL
LIN {X 0,Y 212.27,Z 645.463,A -85,B 0,C 180,E1 -24859.334,E2 -24859.334} C_VEL
LIN {X 0,Y 212.104,Z 650.621,A -85,B 0,C 180,E1 -24862.397,E2 -24862.397} C_VEL
LIN {X 0,Y 211.454,Z 658.391,A -85,B 0,C 180,E1 -24866.19,E2 -24866.19} C_VEL
LIN {X 0,Y 211.237,Z 659.588,A -85,B 0,C 180,E1 -24866.687,E2 -24866.687} C_VEL
LIN {X 0,Y 207.898,Z 667.515,A -85,B 0,C 180,E1 -24868.748,E2 -24868.748} C_VEL
LIN {X 0,Y 204.111,Z 675.01,A -85,B 0,C 180,E1 -24870.598,E2 -24870.598} C_VEL
LIN {X 0,Y 194.823,Z 687.723,A -85,B 0,C 180,E1 -24873.003,E2 -24873.003} C_VEL
LIN {X 0,Y 184.536,Z 699.982,A -85,B 0,C 180,E1 -24875.977,E2 -24875.977} C_VEL
LIN {X 0,Y 174.939,Z 710.291,A -85,B 0,C 180,E1 -24879.349,E2 -24879.349} C_VEL
LIN {X 0,Y 167.107,Z 717.985,A -85,B 0,C 180,E1 -24882.613,E2 -24882.613} C_VEL
LIN {X 0,Y 158.998,Z 725.544,A -85,B 0,C 180,E1 -24886.759,E2 -24886.759} C_VEL
LIN {X 0,Y 150.206,Z 733.2,A -85,B 0,C 180,E1 -24892.541,E2 -24892.541} C_VEL
LIN {X 0,Y 143.174,Z 739.131,A -85,B 0,C 180,E1 -24898.979,E2 -24898.979} C_VEL
LIN {X 0,Y 138.055,Z 743.442,A -85,B 0,C 180,E1 -24905.971,E2 -24905.971} C_VEL
LIN {X 0,Y 135.41,Z 745.792,A -85,B 0,C 180,E1 -24911.859,E2 -24911.859} C_VEL
LIN {X 0,Y 133.987,Z 747.234,A -85,B 0,C 180,E1 -24917.892,E2 -24917.892} C_VEL
LIN {X 0,Y 133.929,Z 747.669,A -85,B 0,C 180,E1 -24925.568,E2 -24925.568} C_VEL
LIN {X 0,Y 134.208,Z 747.201,A -85,B 0,C 180,E1 -24930.003,E2 -24930.003} C_VEL
LIN {X 0,Y 134.017,Z 745.987,A -85,B 0,C 180,E1 -24934.893,E2 -24934.893} C_VEL
LIN {X 0,Y 134.125,Z 742.86,A -85,B 0,C 180,E1 -24942.102,E2 -24942.102} C_VEL
LIN {X 0,Y 135.489,Z 739.009,A -85,B 0,C 180,E1 -24948.136,E2 -24948.136} C_VEL
LIN {X 0,Y 137.939,Z 734.062,A -85,B 0,C 180,E1 -24954.057,E2 -24954.057} C_VEL
LIN {X 0,Y 139.939,Z 730.702,A -85,B 0,C 180,E1 -24957.298,E2 -24957.298} C_VEL
LIN {X 0,Y 140.694,Z 729.51,A -85,B 0,C 180,E1 -24958.756,E2 -24958.756} C_VEL
LIN {X 0,Y 141.264,Z 728.215,A -85,B 0,C 180,E1 -24961.88,E2 -24961.88} C_VEL
LIN {X 0,Y 142.23,Z 726.523,A -85,B 0,C 180,E1 -24966.677,E2 -24966.677} C_VEL
LIN {X 0,Y 143.937,Z 725.559,A -85,B 0,C 180,E1 -24968.942,E2 -24968.942} C_VEL
LIN {X 0,Y 144.813,Z 725.233,A -85,B 0,C 180,E1 -24969.642,E2 -24969.642} C_VEL
LIN {X 0,Y 155.96,Z 721.68,A -85,B 0,C 180,E1 -24976.141,E2 -24976.141} C_VEL
LIN {X 0,Y 160.417,Z 720.294,A -85,B 0,C 180,E1 -24978.144,E2 -24978.144} C_VEL
LIN {X 0,Y 163.308,Z 719.181,A -85,B 0,C 180,E1 -24979.796,E2 -24979.796} C_VEL
LIN {X 0,Y 151.022,Z 718.386,A -85,B 0,C 180,E1 -24986.054,E2 -24986.054} C_VEL
LIN {X 0,Y 141.142,Z 716.354,A -85,B 0,C 180,E1 -24993.377,E2 -24993.377} C_VEL
LIN {X 0,Y 134.053,Z 712.93,A -85,B 0,C 180,E1 -25001.667,E2 -25001.667} C_VEL
LIN {X 0,Y 130.905,Z 709.82,A -85,B 0,C 180,E1 -25007.6,E2 -25007.6} C_VEL
LIN {X 0,Y 128.389,Z 704.823,A -85,B 0,C 180,E1 -25015.292,E2 -25015.292} C_VEL
LIN {X 0,Y 127.886,Z 698.514,A -85,B 0,C 180,E1 -25023.152,E2 -25023.152} C_VEL
LIN {X 0,Y 128.314,Z 692.21,A -85,B 0,C 180,E1 -25029.62,E2 -25029.62} C_VEL
LIN {X 0,Y 129.795,Z 683.996,A -85,B 0,C 180,E1 -25036.517,E2 -25036.517} C_VEL
LIN {X 0,Y 132.701,Z 674.001,A -85,B 0,C 180,E1 -25043.405,E2 -25043.405} C_VEL
LIN {X 0,Y 136.39,Z 663.699,A -85,B 0,C 180,E1 -25049.178,E2 -25049.178} C_VEL
LIN {X 0,Y 138.102,Z 659.443,A -85,B 0,C 180,E1 -25051.336,E2 -25051.336} C_VEL
LIN {X 0,Y 138.852,Z 659.381,A -85,B 0,C 180,E1 -25052.106,E2 -25052.106} C_VEL
LIN {X 0,Y 140.566,Z 658.818,A -85,B 0,C 180,E1 -25053.367,E2 -25053.367} C_VEL
LIN {X 0,Y 142.624,Z 657.844,A -85,B 0,C 180,E1 -25054.521,E2 -25054.521} C_VEL
LIN {X 0,Y 145.015,Z 656.434,A -85,B 0,C 180,E1 -25055.562,E2 -25055.562} C_VEL
LIN {X 0,Y 149.076,Z 654.857,A -85,B 0,C 180,E1 -25057.799,E2 -25057.799} C_VEL
LIN {X 0,Y 153.777,Z 652.56,A -85,B 0,C 180,E1 -25059.781,E2 -25059.781} C_VEL
LIN {X 0,Y 158.436,Z 650.603,A -85,B 0,C 180,E1 -25061.713,E2 -25061.713} C_VEL
LIN {X 0,Y 166.425,Z 646.327,A -85,B 0,C 180,E1 -25064.171,E2 -25064.171} C_VEL
LIN {X 0,Y 171.672,Z 643.765,A -85,B 0,C 180,E1 -25065.761,E2 -25065.761} C_VEL
LIN {X 0,Y 177.491,Z 640.256,A -85,B 0,C 180,E1 -25067.101,E2 -25067.101} C_VEL
LIN {X 0,Y 181.758,Z 638.144,A -85,B 0,C 180,E1 -25068.186,E2 -25068.186} C_VEL
LIN {X 0,Y 181.623,Z 640.233,A -85,B 0,C 180,E1 -25068.863,E2 -25068.863} C_VEL
LIN {X 0,Y 175.252,Z 653.348,A -85,B 0,C 180,E1 -25071.198,E2 -25071.198} C_VEL
LIN {X 0,Y 169.018,Z 664.516,A -85,B 0,C 180,E1 -25073.66,E2 -25073.66} C_VEL
LIN {X 0,Y 161.663,Z 676.722,A -85,B 0,C 180,E1 -25077.081,E2 -25077.081} C_VEL
LIN {X 0,Y 154.908,Z 687.126,A -85,B 0,C 180,E1 -25080.807,E2 -25080.807} C_VEL
LIN {X 0,Y 147.703,Z 697.245,A -85,B 0,C 180,E1 -25085.393,E2 -25085.393} C_VEL
LIN {X 0,Y 141.535,Z 705.922,A -85,B 0,C 180,E1 -25090.644,E2 -25090.644} C_VEL
LIN {X 0,Y 136.01,Z 713.436,A -85,B 0,C 180,E1 -25096.551,E2 -25096.551} C_VEL
LIN {X 0,Y 132.045,Z 719.079,A -85,B 0,C 180,E1 -25102.35,E2 -25102.35} C_VEL
LIN {X 0,Y 129.779,Z 722.562,A -85,B 0,C 180,E1 -25106.892,E2 -25106.892} C_VEL
LIN {X 0,Y 127.786,Z 726.317,A -85,B 0,C 180,E1 -25113.149,E2 -25113.149} C_VEL
LIN {X 0,Y 126.663,Z 729.009,A -85,B 0,C 180,E1 -25119.578,E2 -25119.578} C_VEL
LIN {X 0,Y 126.452,Z 730.764,A -85,B 0,C 180,E1 -25126.131,E2 -25126.131} C_VEL
LIN {X 0,Y 127.126,Z 731.544,A -85,B 0,C 180,E1 -25132.763,E2 -25132.763} C_VEL
LIN {X 0,Y 128.938,Z 731.305,A -85,B 0,C 180,E1 -25139.373,E2 -25139.373} C_VEL
LIN {X 0,Y 131.982,Z 730.094,A -85,B 0,C 180,E1 -25145.851,E2 -25145.851} C_VEL
LIN {X 0,Y 136.357,Z 727.727,A -85,B 0,C 180,E1 -25152.065,E2 -25152.065} C_VEL
LIN {X 0,Y 142.062,Z 724.287,A -85,B 0,C 180,E1 -25157.903,E2 -25157.903} C_VEL
LIN {X 0,Y 149.058,Z 719.648,A -85,B 0,C 180,E1 -25163.271,E2 -25163.271} C_VEL
LIN {X 0,Y 157.168,Z 713.654,A -85,B 0,C 180,E1 -25168.163,E2 -25168.163} C_VEL
LIN {X 0,Y 166.281,Z 706.25,A -85,B 0,C 180,E1 -25172.564,E2 -25172.564} C_VEL
LIN {X 0,Y 176.078,Z 697.36,A -85,B 0,C 180,E1 -25176.474,E2 -25176.474} C_VEL
LIN {X 0,Y 185.541,Z 687.799,A -85,B 0,C 180,E1 -25179.626,E2 -25179.626} C_VEL
LIN {X 0,Y 195.332,Z 676.582,A -85,B 0,C 180,E1 -25182.442,E2 -25182.442} C_VEL
LIN {X 0,Y 204.05,Z 665.185,A -85,B 0,C 180,E1 -25184.654,E2 -25184.654} C_VEL
LIN {X 0,Y 205.675,Z 662.819,A -85,B 0,C 180,E1 -25185.137,E2 -25185.137} C_VEL
LIN {X 0,Y 206.193,Z 657.934,A -85,B 0,C 180,E1 -25188.198,E2 -25188.198} C_VEL
LIN {X 0,Y 206.349,Z 654.169,A -85,B 0,C 180,E1 -25190.988,E2 -25190.988} C_VEL
LIN {X 0,Y 206.462,Z 650.635,A -85,B 0,C 180,E1 -25194.138,E2 -25194.138} C_VEL
LIN {X 0,Y 206.406,Z 647.304,A -85,B 0,C 180,E1 -25198.048,E2 -25198.048} C_VEL
LIN {X 0,Y 206.557,Z 645.089,A -85,B 0,C 180,E1 -25201.949,E2 -25201.949} C_VEL
LIN {X 0,Y 206.741,Z 644.307,A -85,B 0,C 180,E1 -25203.898,E2 -25203.898} C_VEL
LIN {X 0,Y 206.666,Z 644.536,A -85,B 0,C 180,E1 -25207.817,E2 -25207.817} C_VEL
LIN {X 0,Y 207.004,Z 645.729,A -85,B 0,C 180,E1 -25211.753,E2 -25211.753} C_VEL
LIN {X 0,Y 207.25,Z 646.839,A -85,B 0,C 180,E1 -25213.731,E2 -25213.731} C_VEL
LIN {X 0,Y 207.867,Z 649.956,A -85,B 0,C 180,E1 -25217.715,E2 -25217.715} C_VEL
LIN {X 0,Y 208.121,Z 651.202,A -85,B 0,C 180,E1 -25219.007,E2 -25219.007} C_VEL
LIN {X 0,Y 207.701,Z 655.863,A -85,B 0,C 180,E1 -25221.851,E2 -25221.851} C_VEL
LIN {X 0,Y 206.655,Z 663.103,A -85,B 0,C 180,E1 -25225.509,E2 -25225.509} C_VEL
LIN {X 0,Y 203.198,Z 670.442,A -85,B 0,C 180,E1 -25227.488,E2 -25227.488} C_VEL
LIN {X 0,Y 199.269,Z 677.395,A -85,B 0,C 180,E1 -25229.208,E2 -25229.208} C_VEL
LIN {X 0,Y 190.883,Z 688.225,A -85,B 0,C 180,E1 -25231.25,E2 -25231.25} C_VEL
LIN {X 0,Y 181.73,Z 698.778,A -85,B 0,C 180,E1 -25233.756,E2 -25233.756} C_VEL
LIN {X 0,Y 171.703,Z 709.182,A -85,B 0,C 180,E1 -25237.051,E2 -25237.051} C_VEL
LIN {X 0,Y 162.185,Z 718.127,A -85,B 0,C 180,E1 -25240.813,E2 -25240.813} C_VEL
LIN {X 0,Y 153.838,Z 725.46,A -85,B 0,C 180,E1 -25244.923,E2 -25244.923} C_VEL
LIN {X 0,Y 146.28,Z 731.639,A -85,B 0,C 180,E1 -25249.568,E2 -25249.568} C_VEL
LIN {X 0,Y 139.806,Z 736.711,A -85,B 0,C 180,E1 -25254.687,E2 -25254.687} C_VEL
LIN {X 0,Y 135.744,Z 739.819,A -85,B 0,C 180,E1 -25258.823,E2 -25258.823} C_VEL
LIN {X 0,Y 130.758,Z 743.703,A -85,B 0,C 180,E1 -25266.021,E2 -25266.021} C_VEL
LIN {X 0,Y 127.572,Z 746.244,A -85,B 0,C 180,E1 -25274.015,E2 -25274.015} C_VEL
LIN {X 0,Y 126.711,Z 747.134,A -85,B 0,C 180,E1 -25280.425,E2 -25280.425} C_VEL
LIN {X 0,Y 126.903,Z 747.105,A -85,B 0,C 180,E1 -25286.829,E2 -25286.829} C_VEL
LIN {X 0,Y 127.142,Z 746.701,A -85,B 0,C 180,E1 -25290.003,E2 -25290.003} C_VEL
LIN {X 0,Y 126.937,Z 745.56,A -85,B 0,C 180,E1 -25294.751,E2 -25294.751} C_VEL
LIN {X 0,Y 127.118,Z 742.245,A -85,B 0,C 180,E1 -25302.78,E2 -25302.78} C_VEL
LIN {X 0,Y 128.661,Z 738.319,A -85,B 0,C 180,E1 -25309.135,E2 -25309.135} C_VEL
LIN {X 0,Y 131.37,Z 733.289,A -85,B 0,C 180,E1 -25315.343,E2 -25315.343} C_VEL
LIN {X 0,Y 134.728,Z 728.351,A -85,B 0,C 180,E1 -25320.141,E2 -25320.141} C_VEL
LIN {X 0,Y 142.386,Z 725.967,A -85,B 0,C 180,E1 -25327.841,E2 -25327.841} C_VEL
LIN {X 0,Y 144.813,Z 725.233,A -85,B 0,C 180,E1 -25329.642,E2 -25329.642} C_VEL
LIN {X 0,Y 146.17,Z 724.571,A -85,B 0,C 180,E1 -25331.095,E2 -25331.095} C_VEL
LIN {X 0,Y 148.109,Z 722.358,A -85,B 0,C 180,E1 -25336.223,E2 -25336.223} C_VEL
LIN {X 0,Y 149.931,Z 721.688,A -85,B 0,C 180,E1 -25337.555,E2 -25337.555} C_VEL
LIN {X 0,Y 151.083,Z 721.383,A -85,B 0,C 180,E1 -25338.101,E2 -25338.101} C_VEL
LIN {X 0,Y 153.549,Z 720.349,A -85,B 0,C 180,E1 -25340.151,E2 -25340.151} C_VEL
LIN {X 0,Y 141.542,Z 718.75,A -85,B 0,C 180,E1 -25346.896,E2 -25346.896} C_VEL
LIN {X 0,Y 132.014,Z 715.901,A -85,B 0,C 180,E1 -25354.794,E2 -25354.794} C_VEL
LIN {X 0,Y 125.545,Z 711.638,A -85,B 0,C 180,E1 -25363.747,E2 -25363.747} C_VEL
LIN {X 0,Y 122.15,Z 706.889,A -85,B 0,C 180,E1 -25371.731,E2 -25371.731} C_VEL
LIN {X 0,Y 120.775,Z 700.88,A -85,B 0,C 180,E1 -25380.001,E2 -25380.001} C_VEL
LIN {X 0,Y 120.959,Z 694.97,A -85,B 0,C 180,E1 -25386.675,E2 -25386.675} C_VEL
LIN {X 0,Y 121.875,Z 688.019,A -85,B 0,C 180,E1 -25393.338,E2 -25393.338} C_VEL
LIN {X 0,Y 123.795,Z 679.767,A -85,B 0,C 180,E1 -25399.917,E2 -25399.917} C_VEL
LIN {X 0,Y 127.053,Z 670.113,A -85,B 0,C 180,E1 -25406.267,E2 -25406.267} C_VEL
LIN {X 0,Y 128.009,Z 667.688,A -85,B 0,C 180,E1 -25407.82,E2 -25407.82} C_VEL
LIN {X 0,Y 129.273,Z 667.427,A -85,B 0,C 180,E1 -25409.296,E2 -25409.296} C_VEL
LIN {X 0,Y 138.78,Z 663.407,A -85,B 0,C 180,E1 -25415.619,E2 -25415.619} C_VEL
LIN {X 0,Y 145.503,Z 660.382,A -85,B 0,C 180,E1 -25418.898,E2 -25418.898} C_VEL
LIN {X 0,Y 157.692,Z 655.202,A -85,B 0,C 180,E1 -25423.695,E2 -25423.695} C_VEL
LIN {X 0,Y 165.888,Z 651.07,A -85,B 0,C 180,E1 -25426.074,E2 -25426.074} C_VEL
LIN {X 0,Y 172.912,Z 647.597,A -85,B 0,C 180,E1 -25427.884,E2 -25427.884} C_VEL
LIN {X 0,Y 173.409,Z 648.314,A -85,B 0,C 180,E1 -25428.407,E2 -25428.407} C_VEL
LIN {X 0,Y 166.828,Z 660.359,A -85,B 0,C 180,E1 -25430.806,E2 -25430.806} C_VEL
LIN {X 0,Y 160.143,Z 671.518,A -85,B 0,C 180,E1 -25433.666,E2 -25433.666} C_VEL
LIN {X 0,Y 152.757,Z 682.747,A -85,B 0,C 180,E1 -25437.273,E2 -25437.273} C_VEL
LIN {X 0,Y 145.944,Z 692.385,A -85,B 0,C 180,E1 -25441.21,E2 -25441.21} C_VEL
LIN {X 0,Y 139.654,Z 700.58,A -85,B 0,C 180,E1 -25445.467,E2 -25445.467} C_VEL
LIN {X 0,Y 134.355,Z 707.63,A -85,B 0,C 180,E1 -25450.118,E2 -25450.118} C_VEL
LIN {X 0,Y 129.132,Z 714.391,A -85,B 0,C 180,E1 -25455.82,E2 -25455.82} C_VEL
LIN {X 0,Y 125.014,Z 719.919,A -85,B 0,C 180,E1 -25461.917,E2 -25461.917} C_VEL
LIN {X 0,Y 122.65,Z 723.353,A -85,B 0,C 180,E1 -25466.712,E2 -25466.712} C_VEL
LIN {X 0,Y 120.626,Z 727.001,A -85,B 0,C 180,E1 -25473.336,E2 -25473.336} C_VEL
LIN {X 0,Y 119.514,Z 729.65,A -85,B 0,C 180,E1 -25480.157,E2 -25480.157} C_VEL
LIN {X 0,Y 119.405,Z 731.308,A -85,B 0,C 180,E1 -25487.111,E2 -25487.111} C_VEL
LIN {X 0,Y 120.298,Z 732.042,A -85,B 0,C 180,E1 -25494.135,E2 -25494.135} C_VEL
LIN {X 0,Y 122.411,Z 731.703,A -85,B 0,C 180,E1 -25501.108,E2 -25501.108} C_VEL
LIN {X 0,Y 126.657,Z 730.029,A -85,B 0,C 180,E1 -25509.026,E2 -25509.026} C_VEL
LIN {X 0,Y 132.979,Z 726.772,A -85,B 0,C 180,E1 -25516.601,E2 -25516.601} C_VEL
LIN {X 0,Y 140.873,Z 722.066,A -85,B 0,C 180,E1 -25523.224,E2 -25523.224} C_VEL
LIN {X 0,Y 148.798,Z 716.828,A -85,B 0,C 180,E1 -25528.224,E2 -25528.224} C_VEL
LIN {X 0,Y 159.383,Z 708.963,A -85,B 0,C 180,E1 -25533.463,E2 -25533.463} C_VEL
LIN {X 0,Y 168.023,Z 701.71,A -85,B 0,C 180,E1 -25536.948,E2 -25536.948} C_VEL
LIN {X 0,Y 177.423,Z 693,A -85,B 0,C 180,E1 -25540.173,E2 -25540.173} C_VEL
LIN {X 0,Y 187.33,Z 682.71,A -85,B 0,C 180,E1 -25543.062,E2 -25543.062} C_VEL
LIN {X 0,Y 197.641,Z 670.433,A -85,B 0,C 180,E1 -25545.681,E2 -25545.681} C_VEL
LIN {X 0,Y 200.686,Z 666.396,A -85,B 0,C 180,E1 -25546.384,E2 -25546.384} C_VEL
LIN {X 0,Y 201.242,Z 663.989,A -85,B 0,C 180,E1 -25547.904,E2 -25547.904} C_VEL
LIN {X 0,Y 201.684,Z 660.11,A -85,B 0,C 180,E1 -25550.777,E2 -25550.777} C_VEL
LIN {X 0,Y 202.018,Z 656.529,A -85,B 0,C 180,E1 -25554.008,E2 -25554.008} C_VEL
LIN {X 0,Y 202.206,Z 653.213,A -85,B 0,C 180,E1 -25558.007,E2 -25558.007} C_VEL
LIN {X 0,Y 202.51,Z 650.962,A -85,B 0,C 180,E1 -25561.988,E2 -25561.988} C_VEL
LIN {X 0,Y 202.753,Z 650.175,A -85,B 0,C 180,E1 -25563.974,E2 -25563.974} C_VEL
LIN {X 0,Y 202.715,Z 650.461,A -85,B 0,C 180,E1 -25567.97,E2 -25567.97} C_VEL
LIN {X 0,Y 202.856,Z 650.936,A -85,B 0,C 180,E1 -25569.975,E2 -25569.975} C_VEL
LIN {X 0,Y 203.007,Z 651.774,A -85,B 0,C 180,E1 -25571.988,E2 -25571.988} C_VEL
LIN {X 0,Y 203.417,Z 654.476,A -85,B 0,C 180,E1 -25576.044,E2 -25576.044} C_VEL
LIN {X 0,Y 203.763,Z 656.205,A -85,B 0,C 180,E1 -25578.084,E2 -25578.084} C_VEL
LIN {X 0,Y 203.434,Z 659.165,A -85,B 0,C 180,E1 -25580.209,E2 -25580.209} C_VEL
LIN {X 0,Y 202.35,Z 665.198,A -85,B 0,C 180,E1 -25583.544,E2 -25583.544} C_VEL
LIN {X 0,Y 202.053,Z 666.691,A -85,B 0,C 180,E1 -25584.337,E2 -25584.337} C_VEL
LIN {X 0,Y 198.817,Z 672.918,A -85,B 0,C 180,E1 -25586.055,E2 -25586.055} C_VEL
LIN {X 0,Y 195.806,Z 677.892,A -85,B 0,C 180,E1 -25587.341,E2 -25587.341} C_VEL
LIN {X 0,Y 189.713,Z 685.682,A -85,B 0,C 180,E1 -25588.788,E2 -25588.788} C_VEL
LIN {X 0,Y 179.235,Z 697.56,A -85,B 0,C 180,E1 -25591.483,E2 -25591.483} C_VEL
LIN {X 0,Y 170.018,Z 706.864,A -85,B 0,C 180,E1 -25594.24,E2 -25594.24} C_VEL
LIN {X 0,Y 160.126,Z 715.995,A -85,B 0,C 180,E1 -25597.817,E2 -25597.817} C_VEL
LIN {X 0,Y 151.046,Z 723.667,A -85,B 0,C 180,E1 -25601.892,E2 -25601.892} C_VEL
LIN {X 0,Y 142.757,Z 730.062,A -85,B 0,C 180,E1 -25606.436,E2 -25606.436} C_VEL
LIN {X 0,Y 135.61,Z 735.392,A -85,B 0,C 180,E1 -25611.55,E2 -25611.55} C_VEL
LIN {X 0,Y 129.612,Z 739.565,A -85,B 0,C 180,E1 -25617.169,E2 -25617.169} C_VEL
LIN {X 0,Y 123.93,Z 743.549,A -85,B 0,C 180,E1 -25625.138,E2 -25625.138} C_VEL
LIN {X 0,Y 120.682,Z 745.839,A -85,B 0,C 180,E1 -25633.075,E2 -25633.075} C_VEL
LIN {X 0,Y 119.64,Z 746.694,A -85,B 0,C 180,E1 -25639.854,E2 -25639.854} C_VEL
LIN {X 0,Y 119.811,Z 746.599,A -85,B 0,C 180,E1 -25646.641,E2 -25646.641} C_VEL
LIN {X 0,Y 120.076,Z 746.197,A -85,B 0,C 180,E1 -25650.004,E2 -25650.004} C_VEL
LIN {X 0,Y 119.871,Z 745.106,A -85,B 0,C 180,E1 -25654.668,E2 -25654.668} C_VEL
LIN {X 0,Y 119.785,Z 743.128,A -85,B 0,C 180,E1 -25660.141,E2 -25660.141} C_VEL
LIN {X 0,Y 120.811,Z 739.755,A -85,B 0,C 180,E1 -25666.913,E2 -25666.913} C_VEL
LIN {X 0,Y 123.179,Z 735.207,A -85,B 0,C 180,E1 -25673.543,E2 -25673.543} C_VEL
LIN {X 0,Y 126.99,Z 729.527,A -85,B 0,C 180,E1 -25679.877,E2 -25679.877} C_VEL
LIN {X 0,Y 128.705,Z 727.308,A -85,B 0,C 180,E1 -25681.941,E2 -25681.941} C_VEL
LIN {X 0,Y 138.82,Z 724.683,A -85,B 0,C 180,E1 -25691.162,E2 -25691.162} C_VEL
LIN {X 0,Y 149.931,Z 721.688,A -85,B 0,C 180,E1 -25697.555,E2 -25697.555} C_VEL
LIN {X 0,Y 150.422,Z 721.346,A -85,B 0,C 180,E1 -25698.339,E2 -25698.339} C_VEL
LIN {X 0,Y 149.475,Z 721.021,A -85,B 0,C 180,E1 -25699.389,E2 -25699.389} C_VEL
LIN {X 0,Y 146.619,Z 720.72,A -85,B 0,C 180,E1 -25700.726,E2 -25700.726} C_VEL
LIN {X 0,Y 138.091,Z 720.033,A -85,B 0,C 180,E1 -25703.78,E2 -25703.78} C_VEL
LIN {X 0,Y 137.134,Z 719.825,A -85,B 0,C 180,E1 -25704.322,E2 -25704.322} C_VEL
LIN {X 0,Y 128.657,Z 717.526,A -85,B 0,C 180,E1 -25710.554,E2 -25710.554} C_VEL
LIN {X 0,Y 120.659,Z 713.415,A -85,B 0,C 180,E1 -25719.546,E2 -25719.546} C_VEL
LIN {X 0,Y 116.368,Z 708.876,A -85,B 0,C 180,E1 -25727.798,E2 -25727.798} C_VEL
LIN {X 0,Y 113.993,Z 703.067,A -85,B 0,C 180,E1 -25736.467,E2 -25736.467} C_VEL
LIN {X 0,Y 113.844,Z 695.897,A -85,B 0,C 180,E1 -25745.315,E2 -25745.315} C_VEL
LIN {X 0,Y 114.584,Z 688.993,A -85,B 0,C 180,E1 -25752.398,E2 -25752.398} C_VEL
LIN {X 0,Y 116.727,Z 679.697,A -85,B 0,C 180,E1 -25760.257,E2 -25760.257} C_VEL
LIN {X 0,Y 118.192,Z 675.394,A -85,B 0,C 180,E1 -25763.433,E2 -25763.433} C_VEL
LIN {X 0,Y 118.752,Z 675.307,A -85,B 0,C 180,E1 -25764.475,E2 -25764.475} C_VEL
LIN {X 0,Y 125.078,Z 672.606,A -85,B 0,C 180,E1 -25770.379,E2 -25770.379} C_VEL
LIN {X 0,Y 137.14,Z 667.734,A -85,B 0,C 180,E1 -25777.951,E2 -25777.951} C_VEL
LIN {X 0,Y 154.292,Z 660.832,A -85,B 0,C 180,E1 -25784.914,E2 -25784.914} C_VEL
LIN {X 0,Y 163.848,Z 656.361,A -85,B 0,C 180,E1 -25787.561,E2 -25787.561} C_VEL
LIN {X 0,Y 163.901,Z 657.901,A -85,B 0,C 180,E1 -25788.343,E2 -25788.343} C_VEL
LIN {X 0,Y 156.785,Z 669.565,A -85,B 0,C 180,E1 -25791.127,E2 -25791.127} C_VEL
LIN {X 0,Y 148.977,Z 681.183,A -85,B 0,C 180,E1 -25794.694,E2 -25794.694} C_VEL
LIN {X 0,Y 140.774,Z 692.34,A -85,B 0,C 180,E1 -25799.218,E2 -25799.218} C_VEL
LIN {X 0,Y 134.109,Z 700.614,A -85,B 0,C 180,E1 -25803.545,E2 -25803.545} C_VEL
LIN {X 0,Y 127.722,Z 708.631,A -85,B 0,C 180,E1 -25809.038,E2 -25809.038} C_VEL
LIN {X 0,Y 122.255,Z 715.338,A -85,B 0,C 180,E1 -25815.004,E2 -25815.004} C_VEL
LIN {X 0,Y 117.084,Z 721.99,A -85,B 0,C 180,E1 -25823.101,E2 -25823.101} C_VEL
LIN {X 0,Y 114.376,Z 726.024,A -85,B 0,C 180,E1 -25829.996,E2 -25829.996} C_VEL
LIN {X 0,Y 112.78,Z 729.116,A -85,B 0,C 180,E1 -25837.156,E2 -25837.156} C_VEL
LIN {X 0,Y 112.207,Z 731.182,A -85,B 0,C 180,E1 -25844.505,E2 -25844.505} C_VEL
LIN {X 0,Y 112.797,Z 732.298,A -85,B 0,C 180,E1 -25851.948,E2 -25851.948} C_VEL
LIN {X 0,Y 114.607,Z 732.438,A -85,B 0,C 180,E1 -25859.374,E2 -25859.374} C_VEL
LIN {X 0,Y 117.807,Z 731.523,A -85,B 0,C 180,E1 -25866.62,E2 -25866.62} C_VEL
LIN {X 0,Y 122.519,Z 729.617,A -85,B 0,C 180,E1 -25873.494,E2 -25873.494} C_VEL
LIN {X 0,Y 128.68,Z 726.519,A -85,B 0,C 180,E1 -25879.867,E2 -25879.867} C_VEL
LIN {X 0,Y 136.213,Z 722.284,A -85,B 0,C 180,E1 -25885.636,E2 -25885.636} C_VEL
LIN {X 0,Y 145.567,Z 716.371,A -85,B 0,C 180,E1 -25891.13,E2 -25891.13} C_VEL
LIN {X 0,Y 154.63,Z 709.923,A -85,B 0,C 180,E1 -25895.361,E2 -25895.361} C_VEL
LIN {X 0,Y 163.83,Z 702.606,A -85,B 0,C 180,E1 -25898.903,E2 -25898.903} C_VEL
LIN {X 0,Y 173.555,Z 693.998,A -85,B 0,C 180,E1 -25902.094,E2 -25902.094} C_VEL
LIN {X 0,Y 183.773,Z 683.79,A -85,B 0,C 180,E1 -25904.923,E2 -25904.923} C_VEL
LIN {X 0,Y 193.32,Z 672.862,A -85,B 0,C 180,E1 -25907.253,E2 -25907.253} C_VEL
LIN {X 0,Y 195.359,Z 670.406,A -85,B 0,C 180,E1 -25907.71,E2 -25907.71} C_VEL
LIN {X 0,Y 196.157,Z 669.009,A -85,B 0,C 180,E1 -25908.208,E2 -25908.208} C_VEL
LIN {X 0,Y 197.028,Z 664.526,A -85,B 0,C 180,E1 -25911.796,E2 -25911.796} C_VEL
LIN {X 0,Y 197.488,Z 661.148,A -85,B 0,C 180,E1 -25915.126,E2 -25915.126} C_VEL
LIN {X 0,Y 197.822,Z 658.981,A -85,B 0,C 180,E1 -25917.963,E2 -25917.963} C_VEL
LIN {X 0,Y 198.271,Z 656.682,A -85,B 0,C 180,E1 -25922.03,E2 -25922.03} C_VEL
LIN {X 0,Y 198.587,Z 655.922,A -85,B 0,C 180,E1 -25924.058,E2 -25924.058} C_VEL
LIN {X 0,Y 198.582,Z 656.269,A -85,B 0,C 180,E1 -25928.137,E2 -25928.137} C_VEL
LIN {X 0,Y 198.71,Z 656.792,A -85,B 0,C 180,E1 -25930.185,E2 -25930.185} C_VEL
LIN {X 0,Y 198.941,Z 658.954,A -85,B 0,C 180,E1 -25934.316,E2 -25934.316} C_VEL
LIN {X 0,Y 199.259,Z 661.688,A -85,B 0,C 180,E1 -25937.776,E2 -25937.776} C_VEL
LIN {X 0,Y 198.881,Z 664.211,A -85,B 0,C 180,E1 -25939.615,E2 -25939.615} C_VEL
LIN {X 0,Y 197.416,Z 670.147,A -85,B 0,C 180,E1 -25943.053,E2 -25943.053} C_VEL
LIN {X 0,Y 195.913,Z 672.964,A -85,B 0,C 180,E1 -25943.923,E2 -25943.923} C_VEL
LIN {X 0,Y 192.53,Z 678.419,A -85,B 0,C 180,E1 -25945.39,E2 -25945.39} C_VEL
LIN {X 0,Y 189.835,Z 681.95,A -85,B 0,C 180,E1 -25946.14,E2 -25946.14} C_VEL
LIN {X 0,Y 179.835,Z 693.411,A -85,B 0,C 180,E1 -25948.448,E2 -25948.448} C_VEL
LIN {X 0,Y 168.771,Z 704.546,A -85,B 0,C 180,E1 -25951.393,E2 -25951.393} C_VEL
LIN {X 0,Y 158.342,Z 713.922,A -85,B 0,C 180,E1 -25954.809,E2 -25954.809} C_VEL
LIN {X 0,Y 148.652,Z 721.824,A -85,B 0,C 180,E1 -25958.737,E2 -25958.737} C_VEL
LIN {X 0,Y 139.704,Z 728.495,A -85,B 0,C 180,E1 -25963.166,E2 -25963.166} C_VEL
LIN {X 0,Y 131.431,Z 734.21,A -85,B 0,C 180,E1 -25968.469,E2 -25968.469} C_VEL
LIN {X 0,Y 123.603,Z 739.312,A -85,B 0,C 180,E1 -25975.352,E2 -25975.352} C_VEL
LIN {X 0,Y 118.615,Z 742.505,A -85,B 0,C 180,E1 -25981.71,E2 -25981.71} C_VEL
LIN {X 0,Y 115.061,Z 744.683,A -85,B 0,C 180,E1 -25988.505,E2 -25988.505} C_VEL
LIN {X 0,Y 113.023,Z 745.984,A -85,B 0,C 180,E1 -25995.602,E2 -25995.602} C_VEL
LIN {X 0,Y 112.541,Z 746.284,A -85,B 0,C 180,E1 -26002.829,E2 -26002.829} C_VEL
LIN {X 0,Y 112.732,Z 746.094,A -85,B 0,C 180,E1 -26006.43,E2 -26006.43} C_VEL
LIN {X 0,Y 113.008,Z 745.672,A -85,B 0,C 180,E1 -26010.004,E2 -26010.004} C_VEL
LIN {X 0,Y 112.789,Z 744.679,A -85,B 0,C 180,E1 -26014.476,E2 -26014.476} C_VEL
LIN {X 0,Y 112.727,Z 742.51,A -85,B 0,C 180,E1 -26020.784,E2 -26020.784} C_VEL
LIN {X 0,Y 113.956,Z 739.1,A -85,B 0,C 180,E1 -26027.964,E2 -26027.964} C_VEL
LIN {X 0,Y 116.895,Z 733.989,A -85,B 0,C 180,E1 -26035.603,E2 -26035.603} C_VEL
LIN {X 0,Y 120.782,Z 728.705,A -85,B 0,C 180,E1 -26041.584,E2 -26041.584} C_VEL
LIN {X 0,Y 123.201,Z 726.049,A -85,B 0,C 180,E1 -26044.289,E2 -26044.289} C_VEL
LIN {X 0,Y 133.489,Z 723.928,A -85,B 0,C 180,E1 -26053.195,E2 -26053.195} C_VEL
LIN {X 0,Y 143.588,Z 721.628,A -85,B 0,C 180,E1 -26058.901,E2 -26058.901} C_VEL
LIN {X 0,Y 144.693,Z 721.121,A -85,B 0,C 180,E1 -26060.068,E2 -26060.068} C_VEL
LIN {X 0,Y 137.134,Z 719.825,A -85,B 0,C 180,E1 -26064.322,E2 -26064.322} C_VEL
LIN {X 0,Y 133.455,Z 719.186,A -85,B 0,C 180,E1 -26066.256,E2 -26066.256} C_VEL
LIN {X 0,Y 126.275,Z 717.98,A -85,B 0,C 180,E1 -26069.219,E2 -26069.219} C_VEL
LIN {X 0,Y 120.712,Z 716.735,A -85,B 0,C 180,E1 -26071.786,E2 -26071.786} C_VEL
LIN {X 0,Y 117.377,Z 715.626,A -85,B 0,C 180,E1 -26074.072,E2 -26074.072} C_VEL
LIN {X 0,Y 116.542,Z 715.185,A -85,B 0,C 180,E1 -26074.922,E2 -26074.922} C_VEL
LIN {X 0,Y 110.244,Z 709.718,A -85,B 0,C 180,E1 -26085.228,E2 -26085.228} C_VEL
LIN {X 0,Y 107.222,Z 703.893,A -85,B 0,C 180,E1 -26094.359,E2 -26094.359} C_VEL
LIN {X 0,Y 106.683,Z 696.754,A -85,B 0,C 180,E1 -26103.779,E2 -26103.779} C_VEL
LIN {X 0,Y 107.275,Z 689.878,A -85,B 0,C 180,E1 -26111.337,E2 -26111.337} C_VEL
LIN {X 0,Y 108.726,Z 682.841,A -85,B 0,C 180,E1 -26117.883,E2 -26117.883} C_VEL
LIN {X 0,Y 111.15,Z 681.746,A -85,B 0,C 180,E1 -26122.297,E2 -26122.297} C_VEL
LIN {X 0,Y 114.161,Z 680.244,A -85,B 0,C 180,E1 -26125.529,E2 -26125.529} C_VEL
LIN {X 0,Y 120.712,Z 677.64,A -85,B 0,C 180,E1 -26131.602,E2 -26131.602} C_VEL
LIN {X 0,Y 133.225,Z 672.939,A -85,B 0,C 180,E1 -26139.276,E2 -26139.276} C_VEL
LIN {X 0,Y 150.868,Z 666.246,A -85,B 0,C 180,E1 -26146.226,E2 -26146.226} C_VEL
LIN {X 0,Y 153.611,Z 665.15,A -85,B 0,C 180,E1 -26147.059,E2 -26147.059} C_VEL
LIN {X 0,Y 155.072,Z 665.413,A -85,B 0,C 180,E1 -26147.969,E2 -26147.969} C_VEL
LIN {X 0,Y 146.654,Z 677.851,A -85,B 0,C 180,E1 -26151.462,E2 -26151.462} C_VEL
LIN {X 0,Y 138.944,Z 688.293,A -85,B 0,C 180,E1 -26155.313,E2 -26155.313} C_VEL
LIN {X 0,Y 131.601,Z 697.239,A -85,B 0,C 180,E1 -26159.51,E2 -26159.51} C_VEL
LIN {X 0,Y 124.41,Z 705.902,A -85,B 0,C 180,E1 -26164.981,E2 -26164.981} C_VEL
LIN {X 0,Y 118.127,Z 713.094,A -85,B 0,C 180,E1 -26170.896,E2 -26170.896} C_VEL
LIN {X 0,Y 113.029,Z 719.07,A -85,B 0,C 180,E1 -26177.427,E2 -26177.427} C_VEL
LIN {X 0,Y 109.15,Z 723.851,A -85,B 0,C 180,E1 -26184.454,E2 -26184.454} C_VEL
LIN {X 0,Y 107.212,Z 726.756,A -85,B 0,C 180,E1 -26189.996,E2 -26189.996} C_VEL
LIN {X 0,Y 105.596,Z 729.751,A -85,B 0,C 180,E1 -26197.645,E2 -26197.645} C_VEL
LIN {X 0,Y 105.118,Z 731.775,A -85,B 0,C 180,E1 -26205.507,E2 -26205.507} C_VEL
LIN {X 0,Y 105.93,Z 732.795,A -85,B 0,C 180,E1 -26213.453,E2 -26213.453} C_VEL
LIN {X 0,Y 108.104,Z 732.888,A -85,B 0,C 180,E1 -26221.333,E2 -26221.333} C_VEL
LIN {X 0,Y 111.795,Z 731.874,A -85,B 0,C 180,E1 -26228.945,E2 -26228.945} C_VEL
LIN {X 0,Y 117.103,Z 729.863,A -85,B 0,C 180,E1 -26236.064,E2 -26236.064} C_VEL
LIN {X 0,Y 123.878,Z 726.713,A -85,B 0,C 180,E1 -26242.579,E2 -26242.579} C_VEL
LIN {X 0,Y 132.049,Z 722.362,A -85,B 0,C 180,E1 -26248.375,E2 -26248.375} C_VEL
LIN {X 0,Y 141.355,Z 716.784,A -85,B 0,C 180,E1 -26253.492,E2 -26253.492} C_VEL
LIN {X 0,Y 151.601,Z 709.822,A -85,B 0,C 180,E1 -26257.989,E2 -26257.989} C_VEL
LIN {X 0,Y 162.658,Z 701.236,A -85,B 0,C 180,E1 -26261.898,E2 -26261.898} C_VEL
LIN {X 0,Y 172.857,Z 692.23,A -85,B 0,C 180,E1 -26264.921,E2 -26264.921} C_VEL
LIN {X 0,Y 183.49,Z 681.607,A -85,B 0,C 180,E1 -26267.593,E2 -26267.593} C_VEL
LIN {X 0,Y 191.258,Z 672.774,A -85,B 0,C 180,E1 -26269.412,E2 -26269.412} C_VEL
LIN {X 0,Y 192.227,Z 669.004,A -85,B 0,C 180,E1 -26272.647,E2 -26272.647} C_VEL
LIN {X 0,Y 192.884,Z 666.1,A -85,B 0,C 180,E1 -26275.82,E2 -26275.82} C_VEL
LIN {X 0,Y 193.514,Z 663.267,A -85,B 0,C 180,E1 -26279.999,E2 -26279.999} C_VEL
LIN {X 0,Y 194.24,Z 661.55,A -85,B 0,C 180,E1 -26284.149,E2 -26284.149} C_VEL
LIN {X 0,Y 194.275,Z 661.945,A -85,B 0,C 180,E1 -26288.319,E2 -26288.319} C_VEL
LIN {X 0,Y 194.369,Z 662.537,A -85,B 0,C 180,E1 -26290.415,E2 -26290.415} C_VEL
LIN {X 0,Y 194.482,Z 664.828,A -85,B 0,C 180,E1 -26294.652,E2 -26294.652} C_VEL
LIN {X 0,Y 194.576,Z 667.142,A -85,B 0,C 180,E1 -26297.564,E2 -26297.564} C_VEL
LIN {X 0,Y 193.89,Z 669.955,A -85,B 0,C 180,E1 -26299.545,E2 -26299.545} C_VEL
LIN {X 0,Y 192.652,Z 673.947,A -85,B 0,C 180,E1 -26301.957,E2 -26301.957} C_VEL
LIN {X 0,Y 188.199,Z 680.635,A -85,B 0,C 180,E1 -26303.814,E2 -26303.814} C_VEL
LIN {X 0,Y 183.893,Z 685.782,A -85,B 0,C 180,E1 -26304.776,E2 -26304.776} C_VEL
LIN {X 0,Y 172.228,Z 698.079,A -85,B 0,C 180,E1 -26307.441,E2 -26307.441} C_VEL
LIN {X 0,Y 161.04,Z 708.37,A -85,B 0,C 180,E1 -26310.474,E2 -26310.474} C_VEL
LIN {X 0,Y 151.773,Z 716.049,A -85,B 0,C 180,E1 -26313.545,E2 -26313.545} C_VEL
LIN {X 0,Y 141.854,Z 723.601,A -85,B 0,C 180,E1 -26317.567,E2 -26317.567} C_VEL
LIN {X 0,Y 130.582,Z 731.254,A -85,B 0,C 180,E1 -26323.405,E2 -26323.405} C_VEL
LIN {X 0,Y 122.785,Z 736.08,A -85,B 0,C 180,E1 -26328.84,E2 -26328.84} C_VEL
LIN {X 0,Y 114.827,Z 740.726,A -85,B 0,C 180,E1 -26336.58,E2 -26336.58} C_VEL
LIN {X 0,Y 110.158,Z 743.395,A -85,B 0,C 180,E1 -26343.479,E2 -26343.479} C_VEL
LIN {X 0,Y 107.027,Z 745.032,A -85,B 0,C 180,E1 -26350.837,E2 -26350.837} C_VEL
LIN {X 0,Y 105.559,Z 745.818,A -85,B 0,C 180,E1 -26358.483,E2 -26358.483} C_VEL
LIN {X 0,Y 105.65,Z 745.587,A -85,B 0,C 180,E1 -26366.19,E2 -26366.19} C_VEL
LIN {X 0,Y 105.941,Z 745.132,A -85,B 0,C 180,E1 -26370.004,E2 -26370.004} C_VEL
LIN {X 0,Y 105.707,Z 744.252,A -85,B 0,C 180,E1 -26374.246,E2 -26374.246} C_VEL
LIN {X 0,Y 105.703,Z 741.889,A -85,B 0,C 180,E1 -26381.51,E2 -26381.51} C_VEL
LIN {X 0,Y 107.139,Z 738.423,A -85,B 0,C 180,E1 -26389.151,E2 -26389.151} C_VEL
LIN {X 0,Y 110.973,Z 732.558,A -85,B 0,C 180,E1 -26398.156,E2 -26398.156} C_VEL
LIN {X 0,Y 116.929,Z 725.4,A -85,B 0,C 180,E1 -26405.879,E2 -26405.879} C_VEL
LIN {X 0,Y 117.705,Z 724.812,A -85,B 0,C 180,E1 -26406.666,E2 -26406.666} C_VEL
LIN {X 0,Y 128.354,Z 722.989,A -85,B 0,C 180,E1 -26415.386,E2 -26415.386} C_VEL
LIN {X 0,Y 134.423,Z 721.888,A -85,B 0,C 180,E1 -26418.89,E2 -26418.89} C_VEL
LIN {X 0,Y 135.273,Z 721.364,A -85,B 0,C 180,E1 -26420.327,E2 -26420.327} C_VEL
LIN {X 0,Y 122.54,Z 717.975,A -85,B 0,C 180,E1 -26428.926,E2 -26428.926} C_VEL
LIN {X 0,Y 116.542,Z 715.185,A -85,B 0,C 180,E1 -26434.922,E2 -26434.922} C_VEL
LIN {X 0,Y 113.849,Z 713.87,A -85,B 0,C 180,E1 -26437.456,E2 -26437.456} C_VEL
LIN {X 0,Y 108.334,Z 711.399,A -85,B 0,C 180,E1 -26441.513,E2 -26441.513} C_VEL
LIN {X 0,Y 104.181,Z 709.137,A -85,B 0,C 180,E1 -26444.978,E2 -26444.978} C_VEL
LIN {X 0,Y 101.982,Z 707.28,A -85,B 0,C 180,E1 -26447.868,E2 -26447.868} C_VEL
LIN {X 0,Y 101.534,Z 706.619,A -85,B 0,C 180,E1 -26448.891,E2 -26448.891} C_VEL
LIN {X 0,Y 99.637,Z 700.571,A -85,B 0,C 180,E1 -26457.981,E2 -26457.981} C_VEL
LIN {X 0,Y 99.721,Z 694.267,A -85,B 0,C 180,E1 -26466.07,E2 -26466.07} C_VEL
LIN {X 0,Y 100.12,Z 689.993,A -85,B 0,C 180,E1 -26470.911,E2 -26470.911} C_VEL
LIN {X 0,Y 101.722,Z 688.825,A -85,B 0,C 180,E1 -26476.045,E2 -26476.045} C_VEL
LIN {X 0,Y 104.024,Z 687.459,A -85,B 0,C 180,E1 -26479.745,E2 -26479.745} C_VEL
LIN {X 0,Y 106.277,Z 686.49,A -85,B 0,C 180,E1 -26483.379,E2 -26483.379} C_VEL
LIN {X 0,Y 124.614,Z 679.569,A -85,B 0,C 180,E1 -26498.346,E2 -26498.346} C_VEL
LIN {X 0,Y 139.337,Z 674.39,A -85,B 0,C 180,E1 -26504.924,E2 -26504.924} C_VEL
LIN {X 0,Y 144.685,Z 672.456,A -85,B 0,C 180,E1 -26506.772,E2 -26506.772} C_VEL
LIN {X 0,Y 146.1,Z 672.594,A -85,B 0,C 180,E1 -26507.662,E2 -26507.662} C_VEL
LIN {X 0,Y 137.729,Z 683.872,A -85,B 0,C 180,E1 -26511.308,E2 -26511.308} C_VEL
LIN {X 0,Y 129.909,Z 693.542,A -85,B 0,C 180,E1 -26515.383,E2 -26515.383} C_VEL
LIN {X 0,Y 122.573,Z 701.771,A -85,B 0,C 180,E1 -26519.884,E2 -26519.884} C_VEL
LIN {X 0,Y 116.304,Z 708.848,A -85,B 0,C 180,E1 -26524.972,E2 -26524.972} C_VEL
LIN {X 0,Y 109.981,Z 715.632,A -85,B 0,C 180,E1 -26531.363,E2 -26531.363} C_VEL
LIN {X 0,Y 104.967,Z 721.185,A -85,B 0,C 180,E1 -26538.409,E2 -26538.409} C_VEL
LIN {X 0,Y 101.285,Z 725.688,A -85,B 0,C 180,E1 -26546.017,E2 -26546.017} C_VEL
LIN {X 0,Y 98.854,Z 729.575,A -85,B 0,C 180,E1 -26555.52,E2 -26555.52} C_VEL
LIN {X 0,Y 98.066,Z 731.5,A -85,B 0,C 180,E1 -26562.411,E2 -26562.411} C_VEL
LIN {X 0,Y 98.464,Z 732.938,A -85,B 0,C 180,E1 -26570.904,E2 -26570.904} C_VEL
LIN {X 0,Y 100.206,Z 733.417,A -85,B 0,C 180,E1 -26579.398,E2 -26579.398} C_VEL
LIN {X 0,Y 103.627,Z 732.907,A -85,B 0,C 180,E1 -26587.611,E2 -26587.611} C_VEL
LIN {X 0,Y 108.776,Z 731.295,A -85,B 0,C 180,E1 -26595.286,E2 -26595.286} C_VEL
LIN {X 0,Y 115.924,Z 728.453,A -85,B 0,C 180,E1 -26602.679,E2 -26602.679} C_VEL
LIN {X 0,Y 123.638,Z 724.822,A -85,B 0,C 180,E1 -26608.494,E2 -26608.494} C_VEL
LIN {X 0,Y 133.03,Z 719.761,A -85,B 0,C 180,E1 -26613.902,E2 -26613.902} C_VEL
LIN {X 0,Y 143.406,Z 713.401,A -85,B 0,C 180,E1 -26618.604,E2 -26618.604} C_VEL
LIN {X 0,Y 154.616,Z 705.566,A -85,B 0,C 180,E1 -26622.647,E2 -26622.647} C_VEL
LIN {X 0,Y 165.077,Z 697.128,A -85,B 0,C 180,E1 -26625.81,E2 -26625.81} C_VEL
LIN {X 0,Y 175.479,Z 687.67,A -85,B 0,C 180,E1 -26628.447,E2 -26628.447} C_VEL
LIN {X 0,Y 185.2,Z 677.683,A -85,B 0,C 180,E1 -26630.609,E2 -26630.609} C_VEL
LIN {X 0,Y 186.649,Z 675.697,A -85,B 0,C 180,E1 -26631.337,E2 -26631.337} C_VEL
LIN {X 0,Y 187.375,Z 673.444,A -85,B 0,C 180,E1 -26633.538,E2 -26633.538} C_VEL
LIN {X 0,Y 187.92,Z 671.576,A -85,B 0,C 180,E1 -26635.709,E2 -26635.709} C_VEL
LIN {X 0,Y 188.808,Z 668.726,A -85,B 0,C 180,E1 -26639.999,E2 -26639.999} C_VEL
LIN {X 0,Y 189.702,Z 667.029,A -85,B 0,C 180,E1 -26644.248,E2 -26644.248} C_VEL
LIN {X 0,Y 189.739,Z 667.469,A -85,B 0,C 180,E1 -26648.519,E2 -26648.519} C_VEL
LIN {X 0,Y 189.802,Z 668.133,A -85,B 0,C 180,E1 -26650.668,E2 -26650.668} C_VEL
LIN {X 0,Y 189.826,Z 670.566,A -85,B 0,C 180,E1 -26655.019,E2 -26655.019} C_VEL
LIN {X 0,Y 189.707,Z 672.38,A -85,B 0,C 180,E1 -26657.239,E2 -26657.239} C_VEL
LIN {X 0,Y 188.591,Z 675.725,A -85,B 0,C 180,E1 -26659.595,E2 -26659.595} C_VEL
LIN {X 0,Y 187.852,Z 677.658,A -85,B 0,C 180,E1 -26660.73,E2 -26660.73} C_VEL
LIN {X 0,Y 183.992,Z 682.816,A -85,B 0,C 180,E1 -26662.145,E2 -26662.145} C_VEL
LIN {X 0,Y 173.503,Z 693.966,A -85,B 0,C 180,E1 -26664.309,E2 -26664.309} C_VEL
LIN {X 0,Y 161.805,Z 704.848,A -85,B 0,C 180,E1 -26667.081,E2 -26667.081} C_VEL
LIN {X 0,Y 150.639,Z 714.074,A -85,B 0,C 180,E1 -26670.34,E2 -26670.34} C_VEL
LIN {X 0,Y 140.088,Z 721.787,A -85,B 0,C 180,E1 -26674.135,E2 -26674.135} C_VEL
LIN {X 0,Y 130.28,Z 728.262,A -85,B 0,C 180,E1 -26678.543,E2 -26678.543} C_VEL
LIN {X 0,Y 119.99,Z 734.454,A -85,B 0,C 180,E1 -26684.655,E2 -26684.655} C_VEL
LIN {X 0,Y 112.026,Z 738.818,A -85,B 0,C 180,E1 -26691.15,E2 -26691.15} C_VEL
LIN {X 0,Y 106.126,Z 741.848,A -85,B 0,C 180,E1 -26698.014,E2 -26698.014} C_VEL
LIN {X 0,Y 101.788,Z 743.951,A -85,B 0,C 180,E1 -26705.531,E2 -26705.531} C_VEL
LIN {X 0,Y 99.168,Z 745.104,A -85,B 0,C 180,E1 -26713.537,E2 -26713.537} C_VEL
LIN {X 0,Y 98.355,Z 745.335,A -85,B 0,C 180,E1 -26721.788,E2 -26721.788} C_VEL
LIN {X 0,Y 98.576,Z 745.027,A -85,B 0,C 180,E1 -26726.474,E2 -26726.474} C_VEL
LIN {X 0,Y 98.873,Z 744.591,A -85,B 0,C 180,E1 -26730.004,E2 -26730.004} C_VEL
LIN {X 0,Y 98.64,Z 743.798,A -85,B 0,C 180,E1 -26734.09,E2 -26734.09} C_VEL
LIN {X 0,Y 98.68,Z 741.265,A -85,B 0,C 180,E1 -26742.341,E2 -26742.341} C_VEL
LIN {X 0,Y 100.374,Z 737.72,A -85,B 0,C 180,E1 -26750.497,E2 -26750.497} C_VEL
LIN {X 0,Y 103.651,Z 732.975,A -85,B 0,C 180,E1 -26758.34,E2 -26758.34} C_VEL
LIN {X 0,Y 108.79,Z 727.047,A -85,B 0,C 180,E1 -26765.555,E2 -26765.555} C_VEL
LIN {X 0,Y 112.474,Z 723.403,A -85,B 0,C 180,E1 -26769.252,E2 -26769.252} C_VEL
LIN {X 0,Y 126.237,Z 721.573,A -85,B 0,C 180,E1 -26779.38,E2 -26779.38} C_VEL
LIN {X 0,Y 125.872,Z 721.129,A -85,B 0,C 180,E1 -26780.606,E2 -26780.606} C_VEL
LIN {X 0,Y 113.153,Z 716.813,A -85,B 0,C 180,E1 -26790.208,E2 -26790.208} C_VEL
LIN {X 0,Y 105.269,Z 711.535,A -85,B 0,C 180,E1 -26800.501,E2 -26800.501} C_VEL
LIN {X 0,Y 101.534,Z 706.619,A -85,B 0,C 180,E1 -26808.891,E2 -26808.891} C_VEL
LIN {X 0,Y 99.938,Z 704.644,A -85,B 0,C 180,E1 -26811.899,E2 -26811.899} C_VEL
LIN {X 0,Y 93.489,Z 698.323,A -85,B 0,C 180,E1 -26821.041,E2 -26821.041} C_VEL
LIN {X 0,Y 92.702,Z 696.78,A -85,B 0,C 180,E1 -26824.502,E2 -26824.502} C_VEL
LIN {X 0,Y 92.797,Z 696.409,A -85,B 0,C 180,E1 -26825.689,E2 -26825.689} C_VEL
LIN {X 0,Y 94.923,Z 694.281,A -85,B 0,C 180,E1 -26832.835,E2 -26832.835} C_VEL
LIN {X 0,Y 96.453,Z 693.324,A -85,B 0,C 180,E1 -26836.947,E2 -26836.947} C_VEL
LIN {X 0,Y 98.849,Z 692.011,A -85,B 0,C 180,E1 -26840.826,E2 -26840.826} C_VEL
LIN {X 0,Y 101.276,Z 691.003,A -85,B 0,C 180,E1 -26844.607,E2 -26844.607} C_VEL
LIN {X 0,Y 120.473,Z 684.346,A -85,B 0,C 180,E1 -26859.921,E2 -26859.921} C_VEL
LIN {X 0,Y 136.285,Z 679.119,A -85,B 0,C 180,E1 -26866.732,E2 -26866.732} C_VEL
LIN {X 0,Y 135.914,Z 680.681,A -85,B 0,C 180,E1 -26867.758,E2 -26867.758} C_VEL
LIN {X 0,Y 127.573,Z 690.81,A -85,B 0,C 180,E1 -26871.698,E2 -26871.698} C_VEL
LIN {X 0,Y 119.621,Z 699.592,A -85,B 0,C 180,E1 -26876.068,E2 -26876.068} C_VEL
LIN {X 0,Y 111.193,Z 708.591,A -85,B 0,C 180,E1 -26882.349,E2 -26882.349} C_VEL
LIN {X 0,Y 103.302,Z 716.563,A -85,B 0,C 180,E1 -26890.109,E2 -26890.109} C_VEL
LIN {X 0,Y 97.991,Z 722.011,A -85,B 0,C 180,E1 -26897.571,E2 -26897.571} C_VEL
LIN {X 0,Y 94.17,Z 726.412,A -85,B 0,C 180,E1 -26905.715,E2 -26905.715} C_VEL
LIN {X 0,Y 91.77,Z 730.057,A -85,B 0,C 180,E1 -26915.368,E2 -26915.368} C_VEL
LIN {X 0,Y 90.941,Z 732.086,A -85,B 0,C 180,E1 -26923.401,E2 -26923.401} C_VEL
LIN {X 0,Y 91.64,Z 733.542,A -85,B 0,C 180,E1 -26933.025,E2 -26933.025} C_VEL
LIN {X 0,Y 93.74,Z 733.866,A -85,B 0,C 180,E1 -26941.65,E2 -26941.65} C_VEL
LIN {X 0,Y 97.748,Z 733.301,A -85,B 0,C 180,E1 -26950.316,E2 -26950.316} C_VEL
LIN {X 0,Y 103.552,Z 731.597,A -85,B 0,C 180,E1 -26958.286,E2 -26958.286} C_VEL
LIN {X 0,Y 110.968,Z 728.858,A -85,B 0,C 180,E1 -26965.412,E2 -26965.412} C_VEL
LIN {X 0,Y 119.82,Z 724.968,A -85,B 0,C 180,E1 -26971.612,E2 -26971.612} C_VEL
LIN {X 0,Y 129.841,Z 719.792,A -85,B 0,C 180,E1 -26976.941,E2 -26976.941} C_VEL
LIN {X 0,Y 140.804,Z 713.309,A -85,B 0,C 180,E1 -26981.494,E2 -26981.494} C_VEL
LIN {X 0,Y 152.505,Z 705.345,A -85,B 0,C 180,E1 -26985.397,E2 -26985.397} C_VEL
LIN {X 0,Y 163.079,Z 697.085,A -85,B 0,C 180,E1 -26988.319,E2 -26988.319} C_VEL
LIN {X 0,Y 174.541,Z 686.833,A -85,B 0,C 180,E1 -26990.981,E2 -26990.981} C_VEL
LIN {X 0,Y 180.352,Z 681.039,A -85,B 0,C 180,E1 -26992.193,E2 -26992.193} C_VEL
LIN {X 0,Y 181.855,Z 679.328,A -85,B 0,C 180,E1 -26992.784,E2 -26992.784} C_VEL
LIN {X 0,Y 183.035,Z 676.106,A -85,B 0,C 180,E1 -26996.628,E2 -26996.628} C_VEL
LIN {X 0,Y 183.926,Z 674.044,A -85,B 0,C 180,E1 -26999.999,E2 -26999.999} C_VEL
LIN {X 0,Y 184.954,Z 672.309,A -85,B 0,C 180,E1 -27004.358,E2 -27004.358} C_VEL
LIN {X 0,Y 184.989,Z 672.911,A -85,B 0,C 180,E1 -27008.987,E2 -27008.987} C_VEL
LIN {X 0,Y 185.006,Z 673.576,A -85,B 0,C 180,E1 -27010.948,E2 -27010.948} C_VEL
LIN {X 0,Y 184.951,Z 676.132,A -85,B 0,C 180,E1 -27015.425,E2 -27015.425} C_VEL
LIN {X 0,Y 184.813,Z 677.133,A -85,B 0,C 180,E1 -27016.607,E2 -27016.607} C_VEL
LIN {X 0,Y 183.766,Z 679.653,A -85,B 0,C 180,E1 -27018.519,E2 -27018.519} C_VEL
LIN {X 0,Y 183.412,Z 680.422,A -85,B 0,C 180,E1 -27019.02,E2 -27019.02} C_VEL
LIN {X 0,Y 182.546,Z 681.755,A -85,B 0,C 180,E1 -27019.583,E2 -27019.583} C_VEL
LIN {X 0,Y 179.904,Z 684.96,A -85,B 0,C 180,E1 -27020.362,E2 -27020.362} C_VEL
LIN {X 0,Y 169.191,Z 695.734,A -85,B 0,C 180,E1 -27022.454,E2 -27022.454} C_VEL
LIN {X 0,Y 158.682,Z 705.009,A -85,B 0,C 180,E1 -27024.785,E2 -27024.785} C_VEL
LIN {X 0,Y 147.147,Z 714.115,A -85,B 0,C 180,E1 -27027.929,E2 -27027.929} C_VEL
LIN {X 0,Y 136.176,Z 721.777,A -85,B 0,C 180,E1 -27031.626,E2 -27031.626} C_VEL
LIN {X 0,Y 125.917,Z 728.155,A -85,B 0,C 180,E1 -27035.978,E2 -27035.978} C_VEL
LIN {X 0,Y 116.583,Z 733.473,A -85,B 0,C 180,E1 -27041.109,E2 -27041.109} C_VEL
LIN {X 0,Y 106.51,Z 738.573,A -85,B 0,C 180,E1 -27048.718,E2 -27048.718} C_VEL
LIN {X 0,Y 100.073,Z 741.522,A -85,B 0,C 180,E1 -27055.823,E2 -27055.823} C_VEL
LIN {X 0,Y 95.285,Z 743.589,A -85,B 0,C 180,E1 -27063.739,E2 -27063.739} C_VEL
LIN {X 0,Y 92.291,Z 744.664,A -85,B 0,C 180,E1 -27072.271,E2 -27072.271} C_VEL
LIN {X 0,Y 91.281,Z 744.861,A -85,B 0,C 180,E1 -27081.147,E2 -27081.147} C_VEL
LIN {X 0,Y 91.514,Z 744.478,A -85,B 0,C 180,E1 -27086.69,E2 -27086.69} C_VEL
LIN {X 0,Y 91.78,Z 744.048,A -85,B 0,C 180,E1 -27090.005,E2 -27090.005} C_VEL
LIN {X 0,Y 91.542,Z 743.223,A -85,B 0,C 180,E1 -27094.408,E2 -27094.408} C_VEL
LIN {X 0,Y 91.696,Z 740.643,A -85,B 0,C 180,E1 -27103.298,E2 -27103.298} C_VEL
LIN {X 0,Y 93.647,Z 737.013,A -85,B 0,C 180,E1 -27112.044,E2 -27112.044} C_VEL
LIN {X 0,Y 97.355,Z 732.226,A -85,B 0,C 180,E1 -27120.358,E2 -27120.358} C_VEL
LIN {X 0,Y 103.012,Z 726.211,A -85,B 0,C 180,E1 -27127.886,E2 -27127.886} C_VEL
LIN {X 0,Y 107.511,Z 721.979,A -85,B 0,C 180,E1 -27132.075,E2 -27132.075} C_VEL
LIN {X 0,Y 117.168,Z 721.014,A -85,B 0,C 180,E1 -27139.342,E2 -27139.342} C_VEL
LIN {X 0,Y 116.675,Z 720.49,A -85,B 0,C 180,E1 -27140.786,E2 -27140.786} C_VEL
LIN {X 0,Y 107.066,Z 716.816,A -85,B 0,C 180,E1 -27148.325,E2 -27148.325} C_VEL
LIN {X 0,Y 98.631,Z 711.223,A -85,B 0,C 180,E1 -27159.13,E2 -27159.13} C_VEL
LIN {X 0,Y 94.632,Z 706.16,A -85,B 0,C 180,E1 -27167.97,E2 -27167.97} C_VEL
LIN {X 0,Y 92.594,Z 699.777,A -85,B 0,C 180,E1 -27177.827,E2 -27177.827} C_VEL
LIN {X 0,Y 92.448,Z 697.563,A -85,B 0,C 180,E1 -27181.091,E2 -27181.091} C_VEL
LIN {X 0,Y 92.797,Z 696.409,A -85,B 0,C 180,E1 -27185.689,E2 -27185.689} C_VEL
LIN {X 0,Y 93.072,Z 695.819,A -85,B 0,C 180,E1 -27189.302,E2 -27189.302} C_VEL
LIN {X 0,Y 92.931,Z 695.91,A -85,B 0,C 180,E1 -27195.398,E2 -27195.398} C_VEL
LIN {X 0,Y 93.4,Z 696.112,A -85,B 0,C 180,E1 -27200.282,E2 -27200.282} C_VEL
LIN {X 0,Y 94.713,Z 695.84,A -85,B 0,C 180,E1 -27203.799,E2 -27203.799} C_VEL
LIN {X 0,Y 95.403,Z 695.604,A -85,B 0,C 180,E1 -27204.906,E2 -27204.906} C_VEL
LIN {X 0,Y 111.629,Z 690.297,A -85,B 0,C 180,E1 -27219.022,E2 -27219.022} C_VEL
LIN {X 0,Y 126.477,Z 685.796,A -85,B 0,C 180,E1 -27226.253,E2 -27226.253} C_VEL
LIN {X 0,Y 127.273,Z 685.541,A -85,B 0,C 180,E1 -27226.547,E2 -27226.547} C_VEL
LIN {X 0,Y 126.718,Z 686.925,A -85,B 0,C 180,E1 -27227.494,E2 -27227.494} C_VEL
LIN {X 0,Y 117.287,Z 697.152,A -85,B 0,C 180,E1 -27232.103,E2 -27232.103} C_VEL
LIN {X 0,Y 109.566,Z 705.056,A -85,B 0,C 180,E1 -27236.956,E2 -27236.956} C_VEL
LIN {X 0,Y 101.769,Z 712.617,A -85,B 0,C 180,E1 -27243.324,E2 -27243.324} C_VEL
LIN {X 0,Y 95.131,Z 718.887,A -85,B 0,C 180,E1 -27250.578,E2 -27250.578} C_VEL
LIN {X 0,Y 89.889,Z 724.045,A -85,B 0,C 180,E1 -27258.723,E2 -27258.723} C_VEL
LIN {X 0,Y 87.026,Z 727.137,A -85,B 0,C 180,E1 -27265.363,E2 -27265.363} C_VEL
LIN {X 0,Y 84.684,Z 730.534,A -85,B 0,C 180,E1 -27275.171,E2 -27275.171} C_VEL
LIN {X 0,Y 83.837,Z 732.674,A -85,B 0,C 180,E1 -27284.56,E2 -27284.56} C_VEL
LIN {X 0,Y 84.758,Z 734.029,A -85,B 0,C 180,E1 -27294.488,E2 -27294.488} C_VEL
LIN {X 0,Y 87.414,Z 734.319,A -85,B 0,C 180,E1 -27304.243,E2 -27304.243} C_VEL
LIN {X 0,Y 92.099,Z 733.658,A -85,B 0,C 180,E1 -27313.369,E2 -27313.369} C_VEL
LIN {X 0,Y 98.639,Z 731.902,A -85,B 0,C 180,E1 -27321.597,E2 -27321.597} C_VEL
LIN {X 0,Y 106.805,Z 729.058,A -85,B 0,C 180,E1 -27328.798,E2 -27328.798} C_VEL
LIN {X 0,Y 116.573,Z 725.009,A -85,B 0,C 180,E1 -27335.036,E2 -27335.036} C_VEL
LIN {X 0,Y 128.978,Z 718.829,A -85,B 0,C 180,E1 -27340.915,E2 -27340.915} C_VEL
LIN {X 0,Y 140.435,Z 712.086,A -85,B 0,C 180,E1 -27345.096,E2 -27345.096} C_VEL
LIN {X 0,Y 150.768,Z 705.135,A -85,B 0,C 180,E1 -27348.194,E2 -27348.194} C_VEL
LIN {X 0,Y 161.875,Z 696.673,A -85,B 0,C 180,E1 -27350.99,E2 -27350.99} C_VEL
LIN {X 0,Y 173.318,Z 686.578,A -85,B 0,C 180,E1 -27353.409,E2 -27353.409} C_VEL
LIN {X 0,Y 176.638,Z 683.359,A -85,B 0,C 180,E1 -27354.061,E2 -27354.061} C_VEL
LIN {X 0,Y 177.37,Z 682.046,A -85,B 0,C 180,E1 -27355.454,E2 -27355.454} C_VEL
LIN {X 0,Y 178.174,Z 680.454,A -85,B 0,C 180,E1 -27357.738,E2 -27357.738} C_VEL
LIN {X 0,Y 179.455,Z 678.154,A -85,B 0,C 180,E1 -27362.243,E2 -27362.243} C_VEL
LIN {X 0,Y 180.051,Z 677.441,A -85,B 0,C 180,E1 -27364.476,E2 -27364.476} C_VEL
LIN {X 0,Y 180.075,Z 678.068,A -85,B 0,C 180,E1 -27368.98,E2 -27368.98} C_VEL
LIN {X 0,Y 179.967,Z 679.494,A -85,B 0,C 180,E1 -27372.516,E2 -27372.516} C_VEL
LIN {X 0,Y 179.757,Z 681.625,A -85,B 0,C 180,E1 -27375.882,E2 -27375.882} C_VEL
LIN {X 0,Y 178.952,Z 683.445,A -85,B 0,C 180,E1 -27377.352,E2 -27377.352} C_VEL
LIN {X 0,Y 177.523,Z 685.338,A -85,B 0,C 180,E1 -27378.179,E2 -27378.179} C_VEL
LIN {X 0,Y 166.605,Z 696.034,A -85,B 0,C 180,E1 -27380.194,E2 -27380.194} C_VEL
LIN {X 0,Y 154.316,Z 706.404,A -85,B 0,C 180,E1 -27382.752,E2 -27382.752} C_VEL
LIN {X 0,Y 142.479,Z 715.178,A -85,B 0,C 180,E1 -27385.823,E2 -27385.823} C_VEL
LIN {X 0,Y 132.545,Z 721.772,A -85,B 0,C 180,E1 -27388.977,E2 -27388.977} C_VEL
LIN {X 0,Y 119.273,Z 729.495,A -85,B 0,C 180,E1 -27394.426,E2 -27394.426} C_VEL
LIN {X 0,Y 108.99,Z 734.7,A -85,B 0,C 180,E1 -27400.151,E2 -27400.151} C_VEL
LIN {X 0,Y 101.192,Z 738.326,A -85,B 0,C 180,E1 -27406.017,E2 -27406.017} C_VEL
LIN {X 0,Y 94.189,Z 741.199,A -85,B 0,C 180,E1 -27413.356,E2 -27413.356} C_VEL
LIN {X 0,Y 88.891,Z 743.223,A -85,B 0,C 180,E1 -27421.687,E2 -27421.687} C_VEL
LIN {X 0,Y 85.467,Z 744.225,A -85,B 0,C 180,E1 -27430.802,E2 -27430.802} C_VEL
LIN {X 0,Y 84.216,Z 744.386,A -85,B 0,C 180,E1 -27440.397,E2 -27440.397} C_VEL
LIN {X 0,Y 84.448,Z 743.921,A -85,B 0,C 180,E1 -27447.007,E2 -27447.007} C_VEL
LIN {X 0,Y 84.69,Z 743.502,A -85,B 0,C 180,E1 -27450.005,E2 -27450.005} C_VEL
LIN {X 0,Y 84.425,Z 742.636,A -85,B 0,C 180,E1 -27454.78,E2 -27454.78} C_VEL
LIN {X 0,Y 84.72,Z 740.012,A -85,B 0,C 180,E1 -27464.416,E2 -27464.416} C_VEL
LIN {X 0,Y 87.863,Z 735.195,A -85,B 0,C 180,E1 -27476.105,E2 -27476.105} C_VEL
LIN {X 0,Y 92.551,Z 730.028,A -85,B 0,C 180,E1 -27484.722,E2 -27484.722} C_VEL
LIN {X 0,Y 99.291,Z 723.706,A -85,B 0,C 180,E1 -27492.26,E2 -27492.26} C_VEL
LIN {X 0,Y 103.086,Z 720.341,A -85,B 0,C 180,E1 -27495.369,E2 -27495.369} C_VEL
LIN {X 0,Y 109.071,Z 719.959,A -85,B 0,C 180,E1 -27499.885,E2 -27499.885} C_VEL
LIN {X 0,Y 97.291,Z 714.714,A -85,B 0,C 180,E1 -27510.102,E2 -27510.102} C_VEL
LIN {X 0,Y 89.876,Z 708.489,A -85,B 0,C 180,E1 -27521.775,E2 -27521.775} C_VEL
LIN {X 0,Y 88.038,Z 706.071,A -85,B 0,C 180,E1 -27526.146,E2 -27526.146} C_VEL
LIN {X 0,Y 86.099,Z 703.693,A -85,B 0,C 180,E1 -27535.32,E2 -27535.32} C_VEL
LIN {X 0,Y 86.409,Z 702.197,A -85,B 0,C 180,E1 -27540.002,E2 -27540.002} C_VEL
LIN {X 0,Y 89.361,Z 698.58,A -85,B 0,C 180,E1 -27553.649,E2 -27553.649} C_VEL
LIN {X 0,Y 91.034,Z 697.595,A -85,B 0,C 180,E1 -27557.99,E2 -27557.99} C_VEL
LIN {X 0,Y 95.403,Z 695.604,A -85,B 0,C 180,E1 -27564.906,E2 -27564.906} C_VEL
LIN {X 0,Y 97.422,Z 695.113,A -85,B 0,C 180,E1 -27568.198,E2 -27568.198} C_VEL
LIN {X 0,Y 103.427,Z 695.241,A -85,B 0,C 180,E1 -27577.783,E2 -27577.783} C_VEL
LIN {X 0,Y 106.559,Z 694.757,A -85,B 0,C 180,E1 -27580.486,E2 -27580.486} C_VEL
LIN {X 0,Y 107.809,Z 694.437,A -85,B 0,C 180,E1 -27581.275,E2 -27581.275} C_VEL
LIN {X 0,Y 117.869,Z 691.651,A -85,B 0,C 180,E1 -27586.281,E2 -27586.281} C_VEL
LIN {X 0,Y 117.317,Z 692.782,A -85,B 0,C 180,E1 -27587.17,E2 -27587.17} C_VEL
LIN {X 0,Y 108.171,Z 701.81,A -85,B 0,C 180,E1 -27591.882,E2 -27591.882} C_VEL
LIN {X 0,Y 100.236,Z 709.388,A -85,B 0,C 180,E1 -27597.475,E2 -27597.475} C_VEL
LIN {X 0,Y 91.809,Z 716.827,A -85,B 0,C 180,E1 -27605.096,E2 -27605.096} C_VEL
LIN {X 0,Y 85.463,Z 722.422,A -85,B 0,C 180,E1 -27613.268,E2 -27613.268} C_VEL
LIN {X 0,Y 81.767,Z 725.886,A -85,B 0,C 180,E1 -27620.096,E2 -27620.096} C_VEL
LIN {X 0,Y 78.481,Z 729.597,A -85,B 0,C 180,E1 -27629.995,E2 -27629.995} C_VEL
LIN {X 0,Y 77.543,Z 731.083,A -85,B 0,C 180,E1 -27635.194,E2 -27635.194} C_VEL
LIN {X 0,Y 76.749,Z 733.262,A -85,B 0,C 180,E1 -27645.939,E2 -27645.939} C_VEL
LIN {X 0,Y 78.027,Z 734.539,A -85,B 0,C 180,E1 -27656.76,E2 -27656.76} C_VEL
LIN {X 0,Y 81.319,Z 734.769,A -85,B 0,C 180,E1 -27667.22,E2 -27667.22} C_VEL
LIN {X 0,Y 86.722,Z 734.013,A -85,B 0,C 180,E1 -27676.825,E2 -27676.825} C_VEL
LIN {X 0,Y 94.086,Z 732.208,A -85,B 0,C 180,E1 -27685.243,E2 -27685.243} C_VEL
LIN {X 0,Y 103.055,Z 729.259,A -85,B 0,C 180,E1 -27692.434,E2 -27692.434} C_VEL
LIN {X 0,Y 113.358,Z 725.199,A -85,B 0,C 180,E1 -27698.419,E2 -27698.419} C_VEL
LIN {X 0,Y 125.556,Z 719.428,A -85,B 0,C 180,E1 -27703.746,E2 -27703.746} C_VEL
LIN {X 0,Y 139.424,Z 711.559,A -85,B 0,C 180,E1 -27708.366,E2 -27708.366} C_VEL
LIN {X 0,Y 151.605,Z 703.37,A -85,B 0,C 180,E1 -27711.598,E2 -27711.598} C_VEL
LIN {X 0,Y 162.527,Z 694.951,A -85,B 0,C 180,E1 -27713.994,E2 -27713.994} C_VEL
LIN {X 0,Y 170.232,Z 688.298,A -85,B 0,C 180,E1 -27715.48,E2 -27715.48} C_VEL
LIN {X 0,Y 172.07,Z 686.602,A -85,B 0,C 180,E1 -27715.939,E2 -27715.939} C_VEL
LIN {X 0,Y 172.762,Z 685.442,A -85,B 0,C 180,E1 -27717.668,E2 -27717.668} C_VEL
LIN {X 0,Y 173.542,Z 684.126,A -85,B 0,C 180,E1 -27719.999,E2 -27719.999} C_VEL
LIN {X 0,Y 174.284,Z 683.131,A -85,B 0,C 180,E1 -27722.31,E2 -27722.31} C_VEL
LIN {X 0,Y 175.003,Z 682.418,A -85,B 0,C 180,E1 -27724.606,E2 -27724.606} C_VEL
LIN {X 0,Y 174.987,Z 683.156,A -85,B 0,C 180,E1 -27729.244,E2 -27729.244} C_VEL
LIN {X 0,Y 174.891,Z 684.019,A -85,B 0,C 180,E1 -27731.59,E2 -27731.59} C_VEL
LIN {X 0,Y 174.566,Z 685.916,A -85,B 0,C 180,E1 -27734.944,E2 -27734.944} C_VEL
LIN {X 0,Y 174.305,Z 686.55,A -85,B 0,C 180,E1 -27735.636,E2 -27735.636} C_VEL
LIN {X 0,Y 173.489,Z 687.7,A -85,B 0,C 180,E1 -27736.319,E2 -27736.319} C_VEL
LIN {X 0,Y 161.119,Z 698.991,A -85,B 0,C 180,E1 -27738.437,E2 -27738.437} C_VEL
LIN {X 0,Y 150.147,Z 707.746,A -85,B 0,C 180,E1 -27740.596,E2 -27740.596} C_VEL
LIN {X 0,Y 138.023,Z 716.242,A -85,B 0,C 180,E1 -27743.584,E2 -27743.584} C_VEL
LIN {X 0,Y 126.379,Z 723.377,A -85,B 0,C 180,E1 -27747.165,E2 -27747.165} C_VEL
LIN {X 0,Y 115.365,Z 729.374,A -85,B 0,C 180,E1 -27751.483,E2 -27751.483} C_VEL
LIN {X 0,Y 103.859,Z 734.795,A -85,B 0,C 180,E1 -27757.516,E2 -27757.516} C_VEL
LIN {X 0,Y 96.131,Z 738.05,A -85,B 0,C 180,E1 -27763.03,E2 -27763.03} C_VEL
LIN {X 0,Y 88.492,Z 740.878,A -85,B 0,C 180,E1 -27770.561,E2 -27770.561} C_VEL
LIN {X 0,Y 82.61,Z 742.833,A -85,B 0,C 180,E1 -27779.313,E2 -27779.313} C_VEL
LIN {X 0,Y 78.71,Z 743.786,A -85,B 0,C 180,E1 -27789.08,E2 -27789.08} C_VEL
LIN {X 0,Y 77.166,Z 743.9,A -85,B 0,C 180,E1 -27799.511,E2 -27799.511} C_VEL
LIN {X 0,Y 77.601,Z 742.956,A -85,B 0,C 180,E1 -27810.006,E2 -27810.006} C_VEL
LIN {X 0,Y 77.302,Z 742.046,A -85,B 0,C 180,E1 -27815.222,E2 -27815.222} C_VEL
LIN {X 0,Y 77.793,Z 739.383,A -85,B 0,C 180,E1 -27825.731,E2 -27825.731} C_VEL
LIN {X 0,Y 80.466,Z 735.585,A -85,B 0,C 180,E1 -27835.9,E2 -27835.9} C_VEL
LIN {X 0,Y 85.19,Z 730.693,A -85,B 0,C 180,E1 -27845.28,E2 -27845.28} C_VEL
LIN {X 0,Y 92.066,Z 724.526,A -85,B 0,C 180,E1 -27853.401,E2 -27853.401} C_VEL
LIN {X 0,Y 99.155,Z 718.684,A -85,B 0,C 180,E1 -27859.008,E2 -27859.008} C_VEL
LIN {X 0,Y 99.32,Z 718.307,A -85,B 0,C 180,E1 -27860.445,E2 -27860.445} C_VEL
LIN {X 0,Y 93.372,Z 715.656,A -85,B 0,C 180,E1 -27865.634,E2 -27865.634} C_VEL
LIN {X 0,Y 85.723,Z 712.675,A -85,B 0,C 180,E1 -27875.802,E2 -27875.802} C_VEL
LIN {X 0,Y 82.14,Z 709.929,A -85,B 0,C 180,E1 -27885.129,E2 -27885.129} C_VEL
LIN {X 0,Y 80.141,Z 707.622,A -85,B 0,C 180,E1 -27894.971,E2 -27894.971} C_VEL
LIN {X 0,Y 81.014,Z 705.005,A -85,B 0,C 180,E1 -27904.979,E2 -27904.979} C_VEL
LIN {X 0,Y 83.658,Z 702.637,A -85,B 0,C 180,E1 -27914.6,E2 -27914.6} C_VEL
LIN {X 0,Y 94.592,Z 698.278,A -85,B 0,C 180,E1 -27931.34,E2 -27931.34} C_VEL
LIN {X 0,Y 107.809,Z 694.437,A -85,B 0,C 180,E1 -27941.275,E2 -27941.275} C_VEL
LIN {X 0,Y 108.875,Z 694.53,A -85,B 0,C 180,E1 -27942.426,E2 -27942.426} C_VEL
LIN {X 0,Y 108.986,Z 695.686,A -85,B 0,C 180,E1 -27944.123,E2 -27944.123} C_VEL
LIN {X 0,Y 107.713,Z 697.96,A -85,B 0,C 180,E1 -27946.232,E2 -27946.232} C_VEL
LIN {X 0,Y 105.972,Z 700.021,A -85,B 0,C 180,E1 -27947.748,E2 -27947.748} C_VEL
LIN {X 0,Y 100.435,Z 705.246,A -85,B 0,C 180,E1 -27951.205,E2 -27951.205} C_VEL
LIN {X 0,Y 94.702,Z 710.093,A -85,B 0,C 180,E1 -27954.891,E2 -27954.891} C_VEL
LIN {X 0,Y 85.425,Z 717.75,A -85,B 0,C 180,E1 -27963.091,E2 -27963.091} C_VEL
LIN {X 0,Y 78.676,Z 723.238,A -85,B 0,C 180,E1 -27971.775,E2 -27971.775} C_VEL
LIN {X 0,Y 74.734,Z 726.655,A -85,B 0,C 180,E1 -27979.153,E2 -27979.153} C_VEL
LIN {X 0,Y 71.298,Z 730.268,A -85,B 0,C 180,E1 -27989.994,E2 -27989.994} C_VEL
LIN {X 0,Y 70.304,Z 731.731,A -85,B 0,C 180,E1 -27995.731,E2 -27995.731} C_VEL
LIN {X 0,Y 69.701,Z 733.851,A -85,B 0,C 180,E1 -28007.601,E2 -28007.601} C_VEL
LIN {X 0,Y 71.413,Z 735.038,A -85,B 0,C 180,E1 -28019.469,E2 -28019.469} C_VEL
LIN {X 0,Y 75.441,Z 735.224,A -85,B 0,C 180,E1 -28030.693,E2 -28030.693} C_VEL
LIN {X 0,Y 81.702,Z 734.37,A -85,B 0,C 180,E1 -28040.722,E2 -28040.722} C_VEL
LIN {X 0,Y 89.951,Z 732.514,A -85,B 0,C 180,E1 -28049.243,E2 -28049.243} C_VEL
LIN {X 0,Y 99.75,Z 729.466,A -85,B 0,C 180,E1 -28056.326,E2 -28056.326} C_VEL
LIN {X 0,Y 110.785,Z 725.297,A -85,B 0,C 180,E1 -28062.081,E2 -28062.081} C_VEL
LIN {X 0,Y 122.702,Z 719.907,A -85,B 0,C 180,E1 -28066.815,E2 -28066.815} C_VEL
LIN {X 0,Y 136.915,Z 712.158,A -85,B 0,C 180,E1 -28071.14,E2 -28071.14} C_VEL
LIN {X 0,Y 150.863,Z 703.056,A -85,B 0,C 180,E1 -28074.494,E2 -28074.494} C_VEL
LIN {X 0,Y 163.28,Z 693.512,A -85,B 0,C 180,E1 -28076.884,E2 -28076.884} C_VEL
LIN {X 0,Y 167.168,Z 690.206,A -85,B 0,C 180,E1 -28077.589,E2 -28077.589} C_VEL
LIN {X 0,Y 168.1,Z 688.914,A -85,B 0,C 180,E1 -28079.999,E2 -28079.999} C_VEL
LIN {X 0,Y 168.971,Z 687.94,A -85,B 0,C 180,E1 -28082.383,E2 -28082.383} C_VEL
LIN {X 0,Y 169.786,Z 687.238,A -85,B 0,C 180,E1 -28084.748,E2 -28084.748} C_VEL
LIN {X 0,Y 169.756,Z 687.51,A -85,B 0,C 180,E1 -28087.134,E2 -28087.134} C_VEL
LIN {X 0,Y 169.705,Z 688.089,A -85,B 0,C 180,E1 -28089.534,E2 -28089.534} C_VEL
LIN {X 0,Y 169.396,Z 689.662,A -85,B 0,C 180,E1 -28093.189,E2 -28093.189} C_VEL
LIN {X 0,Y 168.342,Z 691.147,A -85,B 0,C 180,E1 -28094.505,E2 -28094.505} C_VEL
LIN {X 0,Y 155.774,Z 701.87,A -85,B 0,C 180,E1 -28096.53,E2 -28096.53} C_VEL
LIN {X 0,Y 143.053,Z 711.208,A -85,B 0,C 180,E1 -28098.975,E2 -28098.975} C_VEL
LIN {X 0,Y 129.346,Z 719.882,A -85,B 0,C 180,E1 -28102.353,E2 -28102.353} C_VEL
LIN {X 0,Y 117.455,Z 726.414,A -85,B 0,C 180,E1 -28106.174,E2 -28106.174} C_VEL
LIN {X 0,Y 106.304,Z 731.771,A -85,B 0,C 180,E1 -28110.753,E2 -28110.753} C_VEL
LIN {X 0,Y 96.058,Z 735.997,A -85,B 0,C 180,E1 -28116.417,E2 -28116.417} C_VEL
LIN {X 0,Y 86.983,Z 739.312,A -85,B 0,C 180,E1 -28123.358,E2 -28123.358} C_VEL
LIN {X 0,Y 77.719,Z 742.117,A -85,B 0,C 180,E1 -28134.47,E2 -28134.47} C_VEL
LIN {X 0,Y 74.004,Z 743.029,A -85,B 0,C 180,E1 -28141.658,E2 -28141.658} C_VEL
LIN {X 0,Y 70.762,Z 743.469,A -85,B 0,C 180,E1 -28152.672,E2 -28152.672} C_VEL
LIN {X 0,Y 70.081,Z 743.034,A -85,B 0,C 180,E1 -28164.251,E2 -28164.251} C_VEL
LIN {X 0,Y 70.514,Z 742.411,A -85,B 0,C 180,E1 -28170.006,E2 -28170.006} C_VEL
LIN {X 0,Y 70.196,Z 741.458,A -85,B 0,C 180,E1 -28175.752,E2 -28175.752} C_VEL
LIN {X 0,Y 70.889,Z 738.75,A -85,B 0,C 180,E1 -28187.309,E2 -28187.309} C_VEL
LIN {X 0,Y 74.035,Z 734.866,A -85,B 0,C 180,E1 -28198.342,E2 -28198.342} C_VEL
LIN {X 0,Y 79.419,Z 729.888,A -85,B 0,C 180,E1 -28208.282,E2 -28208.282} C_VEL
LIN {X 0,Y 86.987,Z 723.676,A -85,B 0,C 180,E1 -28216.654,E2 -28216.654} C_VEL
LIN {X 0,Y 91.474,Z 720.08,A -85,B 0,C 180,E1 -28220.208,E2 -28220.208} C_VEL
LIN {X 0,Y 77.798,Z 714.903,A -85,B 0,C 180,E1 -28238.82,E2 -28238.82} C_VEL
LIN {X 0,Y 76.18,Z 713.576,A -85,B 0,C 180,E1 -28243.935,E2 -28243.935} C_VEL
LIN {X 0,Y 74.068,Z 711.359,A -85,B 0,C 180,E1 -28254.558,E2 -28254.558} C_VEL
LIN {X 0,Y 74.987,Z 708.772,A -85,B 0,C 180,E1 -28265.38,E2 -28265.38} C_VEL
LIN {X 0,Y 77.863,Z 706.507,A -85,B 0,C 180,E1 -28275.713,E2 -28275.713} C_VEL
LIN {X 0,Y 93.661,Z 701.161,A -85,B 0,C 180,E1 -28296.893,E2 -28296.893} C_VEL
LIN {X 0,Y 107.956,Z 697.418,A -85,B 0,C 180,E1 -28305.737,E2 -28305.737} C_VEL
LIN {X 0,Y 107.754,Z 698.274,A -85,B 0,C 180,E1 -28306.772,E2 -28306.772} C_VEL
LIN {X 0,Y 99.174,Z 706.14,A -85,B 0,C 180,E1 -28311.674,E2 -28311.674} C_VEL
LIN {X 0,Y 94.702,Z 710.093,A -85,B 0,C 180,E1 -28314.891,E2 -28314.891} C_VEL
LIN {X 0,Y 90.969,Z 712.919,A -85,B 0,C 180,E1 -28317.119,E2 -28317.119} C_VEL
LIN {X 0,Y 83.68,Z 717.214,A -85,B 0,C 180,E1 -28320.522,E2 -28320.522} C_VEL
LIN {X 0,Y 76.55,Z 721.021,A -85,B 0,C 180,E1 -28324.661,E2 -28324.661} C_VEL
LIN {X 0,Y 73.235,Z 723.085,A -85,B 0,C 180,E1 -28328.07,E2 -28328.07} C_VEL
LIN {X 0,Y 67.724,Z 727.425,A -85,B 0,C 180,E1 -28338.015,E2 -28338.015} C_VEL
LIN {X 0,Y 64.114,Z 730.939,A -85,B 0,C 180,E1 -28349.993,E2 -28349.993} C_VEL
LIN {X 0,Y 62.545,Z 733.554,A -85,B 0,C 180,E1 -28362.98,E2 -28362.98} C_VEL
LIN {X 0,Y 64.063,Z 735.308,A -85,B 0,C 180,E1 -28378.636,E2 -28378.636} C_VEL
LIN {X 0,Y 67.104,Z 735.746,A -85,B 0,C 180,E1 -28388.924,E2 -28388.924} C_VEL
LIN {X 0,Y 73.211,Z 735.326,A -85,B 0,C 180,E1 -28400.162,E2 -28400.162} C_VEL
LIN {X 0,Y 81.496,Z 733.882,A -85,B 0,C 180,E1 -28409.573,E2 -28409.573} C_VEL
LIN {X 0,Y 91.922,Z 731.26,A -85,B 0,C 180,E1 -28417.523,E2 -28417.523} C_VEL
LIN {X 0,Y 105.301,Z 726.753,A -85,B 0,C 180,E1 -28424.514,E2 -28424.514} C_VEL
LIN {X 0,Y 119.652,Z 720.646,A -85,B 0,C 180,E1 -28429.849,E2 -28429.849} C_VEL
LIN {X 0,Y 130.961,Z 714.842,A -85,B 0,C 180,E1 -28433.088,E2 -28433.088} C_VEL
LIN {X 0,Y 144.384,Z 706.811,A -85,B 0,C 180,E1 -28436.187,E2 -28436.187} C_VEL
LIN {X 0,Y 156.419,Z 698.396,A -85,B 0,C 180,E1 -28438.469,E2 -28438.469} C_VEL
LIN {X 0,Y 161.646,Z 694.283,A -85,B 0,C 180,E1 -28439.322,E2 -28439.322} C_VEL
LIN {X 0,Y 162.477,Z 693.555,A -85,B 0,C 180,E1 -28439.999,E2 -28439.999} C_VEL
LIN {X 0,Y 163.469,Z 692.577,A -85,B 0,C 180,E1 -28442.463,E2 -28442.463} C_VEL
LIN {X 0,Y 164.355,Z 691.847,A -85,B 0,C 180,E1 -28444.905,E2 -28444.905} C_VEL
LIN {X 0,Y 164.32,Z 692.162,A -85,B 0,C 180,E1 -28447.371,E2 -28447.371} C_VEL
LIN {X 0,Y 164.184,Z 692.904,A -85,B 0,C 180,E1 -28450.11,E2 -28450.11} C_VEL
LIN {X 0,Y 163.971,Z 693.837,A -85,B 0,C 180,E1 -28452.374,E2 -28452.374} C_VEL
LIN {X 0,Y 160.369,Z 696.916,A -85,B 0,C 180,E1 -28453.041,E2 -28453.041} C_VEL
LIN {X 0,Y 147.359,Z 706.889,A -85,B 0,C 180,E1 -28455.045,E2 -28455.045} C_VEL
LIN {X 0,Y 136.098,Z 714.362,A -85,B 0,C 180,E1 -28457.204,E2 -28457.204} C_VEL
LIN {X 0,Y 123.244,Z 721.834,A -85,B 0,C 180,E1 -28460.298,E2 -28460.298} C_VEL
LIN {X 0,Y 111.488,Z 727.766,A -85,B 0,C 180,E1 -28463.94,E2 -28463.94} C_VEL
LIN {X 0,Y 100.01,Z 732.714,A -85,B 0,C 180,E1 -28468.558,E2 -28468.558} C_VEL
LIN {X 0,Y 86.923,Z 737.498,A -85,B 0,C 180,E1 -28476.056,E2 -28476.056} C_VEL
LIN {X 0,Y 77.887,Z 740.241,A -85,B 0,C 180,E1 -28483.8,E2 -28483.8} C_VEL
LIN {X 0,Y 70.583,Z 742.032,A -85,B 0,C 180,E1 -28493.323,E2 -28493.323} C_VEL
LIN {X 0,Y 65.482,Z 742.91,A -85,B 0,C 180,E1 -28504.584,E2 -28504.584} C_VEL
LIN {X 0,Y 63.136,Z 742.873,A -85,B 0,C 180,E1 -28517.144,E2 -28517.144} C_VEL
LIN {X 0,Y 63.426,Z 741.862,A -85,B 0,C 180,E1 -28530.007,E2 -28530.007} C_VEL
LIN {X 0,Y 63.243,Z 739.611,A -85,B 0,C 180,E1 -28542.848,E2 -28542.848} C_VEL
LIN {X 0,Y 65.581,Z 736.26,A -85,B 0,C 180,E1 -28555.389,E2 -28555.389} C_VEL
LIN {X 0,Y 71.111,Z 731.247,A -85,B 0,C 180,E1 -28567.758,E2 -28567.758} C_VEL
LIN {X 0,Y 79.963,Z 724.47,A -85,B 0,C 180,E1 -28578.345,E2 -28578.345} C_VEL
LIN {X 0,Y 82.219,Z 722.823,A -85,B 0,C 180,E1 -28580.3,E2 -28580.3} C_VEL
LIN {X 0,Y 81.187,Z 721.775,A -85,B 0,C 180,E1 -28582.705,E2 -28582.705} C_VEL
LIN {X 0,Y 70.13,Z 717.036,A -85,B 0,C 180,E1 -28602.507,E2 -28602.507} C_VEL
LIN {X 0,Y 67.872,Z 714.845,A -85,B 0,C 180,E1 -28614.059,E2 -28614.059} C_VEL
LIN {X 0,Y 68.831,Z 712.355,A -85,B 0,C 180,E1 -28625.863,E2 -28625.863} C_VEL
LIN {X 0,Y 77.367,Z 708.138,A -85,B 0,C 180,E1 -28647.016,E2 -28647.016} C_VEL
LIN {X 0,Y 88.924,Z 704.962,A -85,B 0,C 180,E1 -28659.221,E2 -28659.221} C_VEL
LIN {X 0,Y 98.633,Z 702.614,A -85,B 0,C 180,E1 -28665.444,E2 -28665.444} C_VEL
LIN {X 0,Y 97.442,Z 704.009,A -85,B 0,C 180,E1 -28666.744,E2 -28666.744} C_VEL
LIN {X 0,Y 88.093,Z 711.777,A -85,B 0,C 180,E1 -28672.923,E2 -28672.923} C_VEL
LIN {X 0,Y 79.173,Z 718.664,A -85,B 0,C 180,E1 -28680.771,E2 -28680.771} C_VEL
LIN {X 0,Y 73.235,Z 723.085,A -85,B 0,C 180,E1 -28688.07,E2 -28688.07} C_VEL
LIN {X 0,Y 70.159,Z 725.077,A -85,B 0,C 180,E1 -28691.789,E2 -28691.789} C_VEL
LIN {X 0,Y 64.093,Z 728.014,A -85,B 0,C 180,E1 -28697.985,E2 -28697.985} C_VEL
LIN {X 0,Y 59.572,Z 730.04,A -85,B 0,C 180,E1 -28703.768,E2 -28703.768} C_VEL
LIN {X 0,Y 57.218,Z 731.385,A -85,B 0,C 180,E1 -28708.955,E2 -28708.955} C_VEL
LIN {X 0,Y 56.76,Z 731.789,A -85,B 0,C 180,E1 -28710.845,E2 -28710.845} C_VEL
LIN {X 0,Y 55.433,Z 734.148,A -85,B 0,C 180,E1 -28724.68,E2 -28724.68} C_VEL
LIN {X 0,Y 57.285,Z 735.743,A -85,B 0,C 180,E1 -28740.813,E2 -28740.813} C_VEL
LIN {X 0,Y 61.432,Z 736.198,A -85,B 0,C 180,E1 -28753.337,E2 -28753.337} C_VEL
LIN {X 0,Y 68.597,Z 735.734,A -85,B 0,C 180,E1 -28765.035,E2 -28765.035} C_VEL
LIN {X 0,Y 77.909,Z 734.193,A -85,B 0,C 180,E1 -28774.419,E2 -28774.419} C_VEL
LIN {X 0,Y 88.778,Z 731.631,A -85,B 0,C 180,E1 -28781.78,E2 -28781.78} C_VEL
LIN {X 0,Y 102.237,Z 727.347,A -85,B 0,C 180,E1 -28788.097,E2 -28788.097} C_VEL
LIN {X 0,Y 113.535,Z 722.868,A -85,B 0,C 180,E1 -28792.031,E2 -28792.031} C_VEL
LIN {X 0,Y 126.865,Z 716.608,A -85,B 0,C 180,E1 -28795.62,E2 -28795.62} C_VEL
LIN {X 0,Y 140.595,Z 708.857,A -85,B 0,C 180,E1 -28798.559,E2 -28798.559} C_VEL
LIN {X 0,Y 152.714,Z 700.764,A -85,B 0,C 180,E1 -28800.677,E2 -28800.677} C_VEL
LIN {X 0,Y 155.708,Z 698.637,A -85,B 0,C 180,E1 -28801.136,E2 -28801.136} C_VEL
LIN {X 0,Y 157.424,Z 697.295,A -85,B 0,C 180,E1 -28801.757,E2 -28801.757} C_VEL
LIN {X 0,Y 158.792,Z 696.284,A -85,B 0,C 180,E1 -28805.077,E2 -28805.077} C_VEL
LIN {X 0,Y 158.725,Z 696.659,A -85,B 0,C 180,E1 -28807.632,E2 -28807.632} C_VEL
LIN {X 0,Y 158.546,Z 697.375,A -85,B 0,C 180,E1 -28810.212,E2 -28810.212} C_VEL
LIN {X 0,Y 157.364,Z 698.426,A -85,B 0,C 180,E1 -28810.742,E2 -28810.742} C_VEL
LIN {X 0,Y 144.013,Z 708.133,A -85,B 0,C 180,E1 -28812.589,E2 -28812.589} C_VEL
LIN {X 0,Y 130.906,Z 716.37,A -85,B 0,C 180,E1 -28814.916,E2 -28814.916} C_VEL
LIN {X 0,Y 118.099,Z 723.258,A -85,B 0,C 180,E1 -28817.81,E2 -28817.81} C_VEL
LIN {X 0,Y 105.701,Z 728.96,A -85,B 0,C 180,E1 -28821.445,E2 -28821.445} C_VEL
LIN {X 0,Y 93.883,Z 733.63,A -85,B 0,C 180,E1 -28826.075,E2 -28826.075} C_VEL
LIN {X 0,Y 82.874,Z 737.224,A -85,B 0,C 180,E1 -28832.013,E2 -28832.013} C_VEL
LIN {X 0,Y 73.062,Z 739.924,A -85,B 0,C 180,E1 -28839.698,E2 -28839.698} C_VEL
LIN {X 0,Y 64.934,Z 741.634,A -85,B 0,C 180,E1 -28849.513,E2 -28849.513} C_VEL
LIN {X 0,Y 59.075,Z 742.474,A -85,B 0,C 180,E1 -28861.593,E2 -28861.593} C_VEL
LIN {X 0,Y 56.172,Z 742.358,A -85,B 0,C 180,E1 -28875.517,E2 -28875.517} C_VEL
LIN {X 0,Y 56.35,Z 741.316,A -85,B 0,C 180,E1 -28890.008,E2 -28890.008} C_VEL
LIN {X 0,Y 56.267,Z 738.975,A -85,B 0,C 180,E1 -28904.474,E2 -28904.474} C_VEL
LIN {X 0,Y 59.165,Z 735.583,A -85,B 0,C 180,E1 -28918.377,E2 -28918.377} C_VEL
LIN {X 0,Y 66.505,Z 729.829,A -85,B 0,C 180,E1 -28932.978,E2 -28932.978} C_VEL
LIN {X 0,Y 73.018,Z 725.263,A -85,B 0,C 180,E1 -28940.362,E2 -28940.362} C_VEL
LIN {X 0,Y 73.971,Z 724.186,A -85,B 0,C 180,E1 -28942.063,E2 -28942.063} C_VEL
LIN {X 0,Y 62.436,Z 719.166,A -85,B 0,C 180,E1 -28966.993,E2 -28966.993} C_VEL
LIN {X 0,Y 63.958,Z 714.709,A -85,B 0,C 180,E1 -28992.698,E2 -28992.698} C_VEL
LIN {X 0,Y 89.213,Z 707.473,A -85,B 0,C 180,E1 -29025.156,E2 -29025.156} C_VEL
LIN {X 0,Y 87.166,Z 709.278,A -85,B 0,C 180,E1 -29026.888,E2 -29026.888} C_VEL
LIN {X 0,Y 77.499,Z 716.39,A -85,B 0,C 180,E1 -29033.875,E2 -29033.875} C_VEL
LIN {X 0,Y 68.977,Z 722.361,A -85,B 0,C 180,E1 -29042.703,E2 -29042.703} C_VEL
LIN {X 0,Y 62.127,Z 727.114,A -85,B 0,C 180,E1 -29053.565,E2 -29053.565} C_VEL
LIN {X 0,Y 58.537,Z 730.013,A -85,B 0,C 180,E1 -29063.097,E2 -29063.097} C_VEL
LIN {X 0,Y 56.76,Z 731.789,A -85,B 0,C 180,E1 -29070.845,E2 -29070.845} C_VEL
LIN {X 0,Y 55.266,Z 732.969,A -85,B 0,C 180,E1 -29076.555,E2 -29076.555} C_VEL
LIN {X 0,Y 52.029,Z 734.623,A -85,B 0,C 180,E1 -29086.408,E2 -29086.408} C_VEL
LIN {X 0,Y 50.251,Z 735.606,A -85,B 0,C 180,E1 -29095.098,E2 -29095.098} C_VEL
LIN {X 0,Y 50.328,Z 736.096,A -85,B 0,C 180,E1 -29101.882,E2 -29101.882} C_VEL
LIN {X 0,Y 50.733,Z 736.204,A -85,B 0,C 180,E1 -29104.087,E2 -29104.087} C_VEL
LIN {X 0,Y 56.181,Z 736.653,A -85,B 0,C 180,E1 -29118.628,E2 -29118.628} C_VEL
LIN {X 0,Y 64.552,Z 736.143,A -85,B 0,C 180,E1 -29130.558,E2 -29130.558} C_VEL
LIN {X 0,Y 74.927,Z 734.507,A -85,B 0,C 180,E1 -29139.697,E2 -29139.697} C_VEL
LIN {X 0,Y 86.695,Z 731.845,A -85,B 0,C 180,E1 -29146.578,E2 -29146.578} C_VEL
LIN {X 0,Y 99.638,Z 727.928,A -85,B 0,C 180,E1 -29151.888,E2 -29151.888} C_VEL
LIN {X 0,Y 112.734,Z 722.922,A -85,B 0,C 180,E1 -29155.853,E2 -29155.853} C_VEL
LIN {X 0,Y 126.512,Z 716.552,A -85,B 0,C 180,E1 -29159.052,E2 -29159.052} C_VEL
LIN {X 0,Y 140.609,Z 708.719,A -85,B 0,C 180,E1 -29161.651,E2 -29161.651} C_VEL
LIN {X 0,Y 150.793,Z 702.055,A -85,B 0,C 180,E1 -29163.208,E2 -29163.208} C_VEL
LIN {X 0,Y 152.525,Z 700.866,A -85,B 0,C 180,E1 -29163.981,E2 -29163.981} C_VEL
LIN {X 0,Y 153.081,Z 700.561,A -85,B 0,C 180,E1 -29165.267,E2 -29165.267} C_VEL
LIN {X 0,Y 152.973,Z 700.997,A -85,B 0,C 180,E1 -29167.921,E2 -29167.921} C_VEL
LIN {X 0,Y 151.617,Z 702.091,A -85,B 0,C 180,E1 -29168.701,E2 -29168.701} C_VEL
LIN {X 0,Y 139.266,Z 710.489,A -85,B 0,C 180,E1 -29170.265,E2 -29170.265} C_VEL
LIN {X 0,Y 125.942,Z 718.21,A -85,B 0,C 180,E1 -29172.448,E2 -29172.448} C_VEL
LIN {X 0,Y 112.873,Z 724.712,A -85,B 0,C 180,E1 -29175.199,E2 -29175.199} C_VEL
LIN {X 0,Y 100.149,Z 730.097,A -85,B 0,C 180,E1 -29178.687,E2 -29178.687} C_VEL
LIN {X 0,Y 86.026,Z 734.988,A -85,B 0,C 180,E1 -29184.107,E2 -29184.107} C_VEL
LIN {X 0,Y 73.812,Z 738.385,A -85,B 0,C 180,E1 -29191.039,E2 -29191.039} C_VEL
LIN {X 0,Y 63.93,Z 740.523,A -85,B 0,C 180,E1 -29199.7,E2 -29199.7} C_VEL
LIN {X 0,Y 55.911,Z 741.749,A -85,B 0,C 180,E1 -29211.071,E2 -29211.071} C_VEL
LIN {X 0,Y 50.617,Z 742.04,A -85,B 0,C 180,E1 -29225.393,E2 -29225.393} C_VEL
LIN {X 0,Y 48.797,Z 741.433,A -85,B 0,C 180,E1 -29241.728,E2 -29241.728} C_VEL
LIN {X 0,Y 49.198,Z 740.685,A -85,B 0,C 180,E1 -29250.837,E2 -29250.837} C_VEL
LIN {X 0,Y 49.366,Z 738.338,A -85,B 0,C 180,E1 -29266.552,E2 -29266.552} C_VEL
LIN {X 0,Y 52.946,Z 734.89,A -85,B 0,C 180,E1 -29282.079,E2 -29282.079} C_VEL
LIN {X 0,Y 61.645,Z 728.909,A -85,B 0,C 180,E1 -29297.831,E2 -29297.831} C_VEL
LIN {X 0,Y 65.397,Z 726.474,A -85,B 0,C 180,E1 -29302.012,E2 -29302.012} C_VEL
LIN {X 0,Y 64.634,Z 725.895,A -85,B 0,C 180,E1 -29304.073,E2 -29304.073} C_VEL
LIN {X 0,Y 56.136,Z 722.164,A -85,B 0,C 180,E1 -29325.503,E2 -29325.503} C_VEL
LIN {X 0,Y 57.754,Z 717.901,A -85,B 0,C 180,E1 -29354.089,E2 -29354.089} C_VEL
LIN {X 0,Y 79.727,Z 711.991,A -85,B 0,C 180,E1 -29384.849,E2 -29384.849} C_VEL
LIN {X 0,Y 69.48,Z 718.898,A -85,B 0,C 180,E1 -29392.626,E2 -29392.626} C_VEL
LIN {X 0,Y 60.7,Z 724.432,A -85,B 0,C 180,E1 -29402.403,E2 -29402.403} C_VEL
LIN {X 0,Y 53.825,Z 728.92,A -85,B 0,C 180,E1 -29414.854,E2 -29414.854} C_VEL
LIN {X 0,Y 49.703,Z 732.278,A -85,B 0,C 180,E1 -29429.991,E2 -29429.991} C_VEL
LIN {X 0,Y 48.375,Z 734.731,A -85,B 0,C 180,E1 -29446.882,E2 -29446.882} C_VEL
LIN {X 0,Y 50.645,Z 736.188,A -85,B 0,C 180,E1 -29463.706,E2 -29463.706} C_VEL
LIN {X 0,Y 50.733,Z 736.204,A -85,B 0,C 180,E1 -29464.087,E2 -29464.087} C_VEL
LIN {X 0,Y 51.909,Z 736.542,A -85,B 0,C 180,E1 -29470.548,E2 -29470.548} C_VEL
LIN {X 0,Y 53.475,Z 736.886,A -85,B 0,C 180,E1 -29481.211,E2 -29481.211} C_VEL
LIN {X 0,Y 55.788,Z 736.946,A -85,B 0,C 180,E1 -29489.222,E2 -29489.222} C_VEL
LIN {X 0,Y 58.799,Z 736.726,A -85,B 0,C 180,E1 -29494.338,E2 -29494.338} C_VEL
LIN {X 0,Y 60.098,Z 736.612,A -85,B 0,C 180,E1 -29495.774,E2 -29495.774} C_VEL
LIN {X 0,Y 72.628,Z 734.823,A -85,B 0,C 180,E1 -29505.366,E2 -29505.366} C_VEL
LIN {X 0,Y 85.247,Z 732.06,A -85,B 0,C 180,E1 -29511.576,E2 -29511.576} C_VEL
LIN {X 0,Y 98.601,Z 728.172,A -85,B 0,C 180,E1 -29516.193,E2 -29516.193} C_VEL
LIN {X 0,Y 113.685,Z 722.482,A -85,B 0,C 180,E1 -29519.998,E2 -29519.998} C_VEL
LIN {X 0,Y 126.616,Z 716.503,A -85,B 0,C 180,E1 -29522.502,E2 -29522.502} C_VEL
LIN {X 0,Y 141.034,Z 708.545,A -85,B 0,C 180,E1 -29524.742,E2 -29524.742} C_VEL
LIN {X 0,Y 146.812,Z 704.938,A -85,B 0,C 180,E1 -29525.493,E2 -29525.493} C_VEL
LIN {X 0,Y 147.198,Z 704.738,A -85,B 0,C 180,E1 -29525.972,E2 -29525.972} C_VEL
LIN {X 0,Y 145.015,Z 706.203,A -85,B 0,C 180,E1 -29526.564,E2 -29526.564} C_VEL
LIN {X 0,Y 131.361,Z 714.603,A -85,B 0,C 180,E1 -29528.229,E2 -29528.229} C_VEL
LIN {X 0,Y 114.527,Z 723.192,A -85,B 0,C 180,E1 -29530.956,E2 -29530.956} C_VEL
LIN {X 0,Y 98.084,Z 729.967,A -85,B 0,C 180,E1 -29534.71,E2 -29534.71} C_VEL
LIN {X 0,Y 82.265,Z 735.089,A -85,B 0,C 180,E1 -29540.009,E2 -29540.009} C_VEL
LIN {X 0,Y 70.368,Z 738.074,A -85,B 0,C 180,E1 -29546.005,E2 -29546.005} C_VEL
LIN {X 0,Y 59.575,Z 740.169,A -85,B 0,C 180,E1 -29554.346,E2 -29554.346} C_VEL
LIN {X 0,Y 50.511,Z 741.311,A -85,B 0,C 180,E1 -29565.931,E2 -29565.931} C_VEL
LIN {X 0,Y 44.179,Z 741.562,A -85,B 0,C 180,E1 -29581.506,E2 -29581.506} C_VEL
LIN {X 0,Y 41.761,Z 740.879,A -85,B 0,C 180,E1 -29600.322,E2 -29600.322} C_VEL
LIN {X 0,Y 42.165,Z 740.211,A -85,B 0,C 180,E1 -29610.01,E2 -29610.01} C_VEL
LIN {X 0,Y 42.529,Z 737.697,A -85,B 0,C 180,E1 -29629.31,E2 -29629.31} C_VEL
LIN {X 0,Y 46.983,Z 734.162,A -85,B 0,C 180,E1 -29646.762,E2 -29646.762} C_VEL
LIN {X 0,Y 56.065,Z 728.687,A -85,B 0,C 180,E1 -29662.067,E2 -29662.067} C_VEL
LIN {X 0,Y 56.699,Z 727.778,A -85,B 0,C 180,E1 -29664.447,E2 -29664.447} C_VEL
LIN {X 0,Y 49.821,Z 724.948,A -85,B 0,C 180,E1 -29683.616,E2 -29683.616} C_VEL
LIN {X 0,Y 51.498,Z 720.832,A -85,B 0,C 180,E1 -29715.843,E2 -29715.843} C_VEL
LIN {X 0,Y 65.366,Z 717.112,A -85,B 0,C 180,E1 -29740.177,E2 -29740.177} C_VEL
LIN {X 0,Y 69.246,Z 716.611,A -85,B 0,C 180,E1 -29744.721,E2 -29744.721} C_VEL
LIN {X 0,Y 59.041,Z 722.662,A -85,B 0,C 180,E1 -29753.466,E2 -29753.466} C_VEL
LIN {X 0,Y 50.4,Z 727.564,A -85,B 0,C 180,E1 -29765.261,E2 -29765.261} C_VEL
LIN {X 0,Y 44.308,Z 731.443,A -85,B 0,C 180,E1 -29780.864,E2 -29780.864} C_VEL
LIN {X 0,Y 42.192,Z 733.236,A -85,B 0,C 180,E1 -29791.781,E2 -29791.781} C_VEL
LIN {X 0,Y 41.402,Z 735.315,A -85,B 0,C 180,E1 -29809.835,E2 -29809.835} C_VEL
LIN {X 0,Y 44.609,Z 736.735,A -85,B 0,C 180,E1 -29829.051,E2 -29829.051} C_VEL
LIN {X 0,Y 53.986,Z 737.074,A -85,B 0,C 180,E1 -29848.615,E2 -29848.615} C_VEL
LIN {X 0,Y 60.098,Z 736.612,A -85,B 0,C 180,E1 -29855.774,E2 -29855.774} C_VEL
LIN {X 0,Y 63.859,Z 736.271,A -85,B 0,C 180,E1 -29859.979,E2 -29859.979} C_VEL
LIN {X 0,Y 69.456,Z 735.514,A -85,B 0,C 180,E1 -29867.004,E2 -29867.004} C_VEL
LIN {X 0,Y 74.44,Z 734.581,A -85,B 0,C 180,E1 -29871.891,E2 -29871.891} C_VEL
LIN {X 0,Y 78.937,Z 733.594,A -85,B 0,C 180,E1 -29874.673,E2 -29874.673} C_VEL
LIN {X 0,Y 80.609,Z 733.2,A -85,B 0,C 180,E1 -29875.369,E2 -29875.369} C_VEL
LIN {X 0,Y 95.801,Z 729.115,A -85,B 0,C 180,E1 -29879.998,E2 -29879.998} C_VEL
LIN {X 0,Y 109.012,Z 724.497,A -85,B 0,C 180,E1 -29882.902,E2 -29882.902} C_VEL
LIN {X 0,Y 123.885,Z 718.102,A -85,B 0,C 180,E1 -29885.448,E2 -29885.448} C_VEL
LIN {X 0,Y 120.219,Z 719.934,A -85,B 0,C 180,E1 -29886.412,E2 -29886.412} C_VEL
LIN {X 0,Y 106.596,Z 726.009,A -85,B 0,C 180,E1 -29888.551,E2 -29888.551} C_VEL
LIN {X 0,Y 89.871,Z 732.006,A -85,B 0,C 180,E1 -29892.199,E2 -29892.199} C_VEL
LIN {X 0,Y 79.435,Z 735.035,A -85,B 0,C 180,E1 -29895.39,E2 -29895.39} C_VEL
LIN {X 0,Y 61.531,Z 738.901,A -85,B 0,C 180,E1 -29903.99,E2 -29903.99} C_VEL
LIN {X 0,Y 49.29,Z 740.589,A -85,B 0,C 180,E1 -29914.769,E2 -29914.769} C_VEL
LIN {X 0,Y 41.385,Z 741.105,A -85,B 0,C 180,E1 -29927.227,E2 -29927.227} C_VEL
LIN {X 0,Y 35.772,Z 740.808,A -85,B 0,C 180,E1 -29946.876,E2 -29946.876} C_VEL
LIN {X 0,Y 35.044,Z 739.626,A -85,B 0,C 180,E1 -29970.012,E2 -29970.012} C_VEL
LIN {X 0,Y 35.842,Z 737.057,A -85,B 0,C 180,E1 -29993.102,E2 -29993.102} C_VEL
LIN {X 0,Y 43.416,Z 732.33,A -85,B 0,C 180,E1 -30016.77,E2 -30016.77} C_VEL
LIN {X 0,Y 48.566,Z 729.588,A -85,B 0,C 180,E1 -30024.635,E2 -30024.635} C_VEL
